C01819=1060.196,-45.835,434.393,171.436,27.271,155.094
C01820=1060.190,-46.085,434.406,171.434,27.269,155.094
C01821=1060.184,-46.335,434.419,171.432,27.267,155.094
C01822=1060.178,-46.584,434.432,171.431,27.265,155.094
C01823=1060.172,-46.833,434.444,171.429,27.263,155.093
C01824=1060.166,-47.083,434.456,171.428,27.261,155.093
C01825=1060.160,-47.332,434.469,171.426,27.259,155.093
C01826=1060.154,-47.582,434.481,171.424,27.257,155.093
C01827=1060.147,-47.831,434.494,171.423,27.255,155.093
C01828=1060.142,-48.081,434.506,171.421,27.254,155.093
C01829=1060.136,-48.331,434.519,171.419,27.251,155.092
C01830=1060.130,-48.581,434.531,171.418,27.250,155.092
C01831=1060.123,-48.831,434.543,171.416,27.247,155.092
C01832=1060.117,-49.080,434.556,171.414,27.246,155.092
C01833=1060.112,-49.330,434.568,171.413,27.244,155.092
C01834=1060.105,-49.579,434.581,171.411,27.242,155.091
C01835=1060.099,-49.828,434.593,171.409,27.240,155.091
C01836=1060.093,-50.108,434.607,171.408,27.238,155.091
C01837=1060.086,-50.387,434.621,171.406,27.236,155.091
C01838=1060.078,-50.667,434.635,171.403,27.234,155.091
C01839=1060.071,-50.946,434.648,171.402,27.232,155.091
C01840=1060.065,-51.195,434.660,171.400,27.230,155.090
C01841=1060.059,-51.444,434.673,171.399,27.228,155.090
C01842=1060.053,-51.694,434.685,171.397,27.227,155.090
C01843=1060.047,-51.944,434.697,171.395,27.225,155.090
C01844=1060.040,-52.193,434.709,171.394,27.223,155.090
C01845=1060.034,-52.443,434.722,171.392,27.221,155.090
C01846=1060.028,-52.693,434.734,171.390,27.219,155.089
C01847=1060.021,-52.942,434.746,171.389,27.218,155.089
C01848=1060.015,-53.192,434.758,171.387,27.216,155.089
C01849=1060.008,-53.442,434.770,171.385,27.214,155.089
C01850=1060.003,-53.691,434.782,171.384,27.213,155.089
C01851=1059.996,-53.941,434.794,171.382,27.211,155.089
C01852=1059.990,-54.190,434.806,171.380,27.209,155.089
C01853=1059.984,-54.440,434.819,171.378,27.207,155.088
C01854=1059.977,-54.690,434.831,171.377,27.206,155.088
C01855=1059.971,-54.940,434.843,171.375,27.203,155.088
C01856=1059.965,-55.189,434.855,171.374,27.202,155.088
C01857=1059.959,-55.438,434.867,171.371,27.200,155.088
C01858=1059.953,-55.688,434.879,171.369,27.198,155.088
C01859=1059.946,-55.938,434.891,171.368,27.196,155.087
C01860=1059.940,-56.188,434.903,171.366,27.195,155.087
C01861=1059.934,-56.437,434.915,171.364,27.193,155.087
C01862=1059.928,-56.686,434.927,171.362,27.191,155.087
C01863=1059.922,-56.936,434.939,171.361,27.190,155.087
C01864=1059.915,-57.186,434.951,171.359,27.188,155.087
C01865=1059.909,-57.435,434.963,171.357,27.186,155.087
C01866=1059.903,-57.686,434.975,171.356,27.184,155.086
C01867=1059.897,-57.935,434.987,171.354,27.183,155.086
C01868=1059.890,-58.184,434.999,171.352,27.181,155.086
C01869=1059.884,-58.434,435.011,171.351,27.179,155.086
C01870=1059.878,-58.684,435.023,171.349,27.178,155.086
C01871=1059.872,-58.933,435.034,171.347,27.176,155.086
C01872=1059.866,-59.183,435.047,171.346,27.174,155.086
C01873=1059.859,-59.433,435.058,171.344,27.172,155.085
C01874=1059.853,-59.682,435.070,171.342,27.171,155.085
C01875=1059.847,-59.931,435.083,171.341,27.169,155.085
C01876=1059.841,-60.182,435.094,171.339,27.167,155.085
C01877=1059.834,-60.431,435.106,171.337,27.166,155.085
C01878=1059.829,-60.681,435.118,171.336,27.164,155.085
C01879=1059.823,-60.930,435.130,171.334,27.162,155.085
C01880=1059.816,-61.180,435.141,171.332,27.161,155.084
C01881=1059.810,-61.430,435.154,171.331,27.159,155.084
C01882=1059.804,-61.680,435.166,171.329,27.157,155.084
C01883=1059.798,-61.929,435.177,171.326,27.155,155.084
C01884=1059.792,-62.179,435.189,171.325,27.153,155.084
C01885=1059.785,-62.429,435.201,171.323,27.152,155.084
C01886=1059.779,-62.677,435.213,171.321,27.150,155.084
C01887=1059.774,-62.928,435.225,171.320,27.148,155.083
C01888=1059.767,-63.178,435.237,171.318,27.147,155.083
C01889=1059.761,-63.426,435.248,171.316,27.145,155.083
C01890=1059.755,-63.677,435.260,171.315,27.143,155.083
C01891=1059.749,-63.926,435.272,171.313,27.141,155.083
C01892=1059.743,-64.175,435.283,171.311,27.140,155.083
C01893=1059.736,-64.426,435.295,171.309,27.138,155.083
C01894=1059.730,-64.675,435.307,171.308,27.136,155.082
C01895=1059.725,-64.925,435.318,171.306,27.135,155.082
C01896=1059.718,-65.174,435.330,171.304,27.134,155.082
C01897=1059.712,-65.424,435.343,171.303,27.132,155.082
C01898=1059.706,-65.674,435.354,171.301,27.130,155.082
C01899=1059.700,-65.923,435.366,171.299,27.128,155.082
C01900=1059.693,-66.204,435.378,171.297,27.126,155.082
C01901=1059.686,-66.484,435.392,171.295,27.125,155.082
C01902=1059.680,-66.765,435.404,171.293,27.123,155.081
C01903=1059.672,-67.045,435.418,171.292,27.121,155.081
C01904=1059.667,-67.295,435.429,171.290,27.120,155.081
C01905=1059.661,-67.545,435.441,171.287,27.118,155.081
C01906=1059.654,-67.794,435.453,171.286,27.116,155.081
C01907=1059.648,-68.044,435.464,171.284,27.114,155.081
C01908=1059.642,-68.293,435.477,171.282,27.112,155.081
C01909=1059.637,-68.543,435.488,171.281,27.111,155.080
C01910=1059.630,-68.793,435.499,171.279,27.109,155.080
C01911=1059.624,-69.042,435.510,171.277,27.107,155.080
C01912=1059.618,-69.292,435.523,171.276,27.106,155.080
C01913=1059.612,-69.542,435.534,171.274,27.104,155.080
C01914=1059.606,-69.791,435.546,171.272,27.103,155.080
C01915=1059.600,-70.041,435.557,171.270,27.101,155.080
C01916=1059.594,-70.291,435.568,171.269,27.099,155.080
C01917=1059.588,-70.541,435.580,171.267,27.098,155.079
C01918=1059.582,-70.790,435.591,171.265,27.097,155.079
C01919=1059.576,-71.040,435.603,171.264,27.095,155.079
C01920=1059.570,-71.289,435.614,171.262,27.093,155.079
C01921=1059.564,-71.539,435.627,171.260,27.091,155.079
C01922=1059.558,-71.788,435.638,171.259,27.090,155.079
C01923=1059.552,-72.039,435.649,171.257,27.089,155.079
C01924=1059.546,-72.288,435.660,171.255,27.087,155.079
C01925=1059.539,-72.538,435.672,171.253,27.085,155.079
C01926=1059.534,-72.787,435.684,171.251,27.083,155.078
C01927=1059.528,-73.037,435.695,171.249,27.082,155.078
C01928=1059.522,-73.287,435.706,171.247,27.080,155.078
C01929=1059.515,-73.536,435.718,171.246,27.079,155.078
C01930=1059.510,-73.786,435.729,171.244,27.077,155.078
C01931=1059.504,-74.036,435.741,171.242,27.076,155.078
C01932=1059.497,-74.285,435.752,171.241,27.074,155.078
C01933=1059.491,-74.535,435.763,171.239,27.072,155.078
C01934=1059.485,-74.784,435.774,171.237,27.071,155.078
C01935=1059.479,-75.034,435.786,171.235,27.070,155.078
C01936=1059.473,-75.283,435.797,171.234,27.068,155.077
C01937=1059.467,-75.534,435.808,171.232,27.067,155.077
C01938=1059.461,-75.783,435.819,171.230,27.065,155.077
C01939=1059.454,-76.033,435.831,171.229,27.064,155.077
C01940=1059.448,-76.282,435.842,171.227,27.062,155.077
C01941=1059.442,-76.532,435.853,171.225,27.061,155.077
C01942=1059.436,-76.782,435.864,171.223,27.059,155.077
C01943=1059.430,-77.031,435.876,171.221,27.057,155.077
C01944=1059.424,-77.281,435.887,171.219,27.056,155.077
C01945=1059.418,-77.531,435.898,171.217,27.054,155.077
C01946=1059.412,-77.781,435.909,171.216,27.053,155.077
C01947=1059.406,-78.031,435.920,171.214,27.052,155.076
C01948=1059.399,-78.280,435.931,171.212,27.051,155.076
C01949=1059.393,-78.530,435.943,171.210,27.049,155.076
C01950=1059.387,-78.779,435.954,171.209,27.048,155.076
C01951=1059.381,-79.030,435.965,171.207,27.046,155.076
C01952=1059.375,-79.279,435.976,171.205,27.045,155.076
C01953=1059.369,-79.528,435.987,171.204,27.043,155.076
C01954=1059.363,-79.778,435.999,171.202,27.042,155.076
C01955=1059.356,-80.027,436.009,171.200,27.040,155.076
C01956=1059.350,-80.277,436.020,171.198,27.039,155.076
C01957=1059.344,-80.527,436.031,171.196,27.037,155.076
C01958=1059.338,-80.777,436.042,171.194,27.036,155.076
C01959=1059.332,-81.026,436.052,171.192,27.035,155.076
C01960=1059.325,-81.277,436.064,171.191,27.033,155.075
C01961=1059.319,-81.526,436.075,171.189,27.032,155.075
C01962=1059.312,-81.776,436.085,171.187,27.031,155.075
C01963=1059.306,-82.025,436.097,171.185,27.029,155.075
C01964=1059.300,-82.308,436.109,171.183,27.028,155.075
C01965=1059.292,-82.590,436.122,171.181,27.026,155.075
C01966=1059.285,-82.873,436.133,171.179,27.025,155.075
C01967=1059.279,-83.156,436.146,171.177,27.023,155.075
C01968=1059.272,-83.405,436.156,171.176,27.022,155.075
C01969=1059.266,-83.655,436.168,171.173,27.021,155.075
C01970=1059.260,-83.905,436.179,171.171,27.019,155.075
C01971=1059.254,-84.154,436.189,171.169,27.018,155.075
C01972=1059.247,-84.404,436.200,171.168,27.017,155.075
C01973=1059.241,-84.654,436.211,171.166,27.015,155.075
C01974=1059.235,-84.904,436.222,171.164,27.014,155.075
C01975=1059.229,-85.153,436.233,171.162,27.013,155.075
C01976=1059.223,-85.403,436.243,171.161,27.012,155.075
C01977=1059.216,-85.653,436.255,171.159,27.010,155.074
C01978=1059.210,-85.902,436.265,171.157,27.009,155.074
C01979=1059.204,-86.152,436.276,171.155,27.008,155.074
C01980=1059.198,-86.402,436.287,171.154,27.007,155.074
C01981=1059.191,-86.651,436.297,171.152,27.005,155.074
C01982=1059.185,-86.901,436.309,171.149,27.004,155.074
C01983=1059.179,-87.151,436.319,171.148,27.002,155.074
C01984=1059.173,-87.400,436.330,171.146,27.001,155.074
C01985=1059.167,-87.651,436.340,171.144,27.000,155.074
C01986=1059.161,-87.900,436.351,171.142,26.998,155.074
C01987=1059.155,-88.149,436.361,171.141,26.997,155.074
C01988=1059.148,-88.399,436.373,171.139,26.996,155.074
C01989=1059.143,-88.649,436.384,171.137,26.994,155.074
C01990=1059.136,-88.898,436.394,171.135,26.993,155.074
C01991=1059.130,-89.148,436.405,171.134,26.992,155.074
C01992=1059.124,-89.398,436.415,171.132,26.991,155.074
C01993=1059.118,-89.648,436.426,171.130,26.990,155.074
C01994=1059.112,-89.897,436.436,171.128,26.989,155.074
C01995=1059.106,-90.147,436.448,171.126,26.987,155.074
C01996=1059.099,-90.396,436.458,171.124,26.986,155.074
C01997=1059.094,-90.646,436.469,171.122,26.985,155.074
C01998=1059.087,-90.896,436.479,171.120,26.983,155.074
C01999=1059.081,-91.146,436.490,171.118,26.982,155.074
C02000=1059.075,-91.395,436.500,171.117,26.981,155.074
C02001=1059.069,-91.645,436.511,171.115,26.980,155.073
C02002=1059.063,-91.895,436.521,171.113,26.978,155.073
C02003=1059.057,-92.145,436.532,171.111,26.977,155.073
C02004=1059.051,-92.394,436.542,171.110,26.976,155.073
C02005=1059.045,-92.644,436.553,171.108,26.975,155.073
C02006=1059.038,-92.894,436.563,171.106,26.974,155.073
C02007=1059.032,-93.144,436.574,171.104,26.973,155.073
C02008=1059.027,-93.393,436.585,171.102,26.971,155.073
C02009=1059.020,-93.642,436.595,171.100,26.970,155.073
C02010=1059.014,-93.893,436.606,171.098,26.969,155.073
C02011=1059.008,-94.142,436.616,171.096,26.967,155.073
C02012=1059.002,-94.392,436.627,171.095,26.966,155.073
C02013=1058.996,-94.642,436.637,171.093,26.965,155.073
C02014=1058.990,-94.891,436.647,171.091,26.964,155.073
C02015=1058.984,-95.141,436.659,171.089,26.963,155.073
C02016=1058.977,-95.391,436.668,171.088,26.962,155.073
C02017=1058.972,-95.640,436.679,171.086,26.961,155.073
C02018=1058.966,-95.890,436.690,171.084,26.959,155.073
C02019=1058.960,-96.140,436.700,171.082,26.958,155.073
C02020=1058.954,-96.389,436.710,171.079,26.957,155.073
C02021=1058.947,-96.639,436.721,171.078,26.956,155.073
C02022=1058.942,-96.889,436.731,171.076,26.955,155.073
C02023=1058.935,-97.138,436.742,171.074,26.954,155.073
C02024=1058.930,-97.388,436.752,171.072,26.952,155.073
C02025=1058.923,-97.638,436.762,171.071,26.951,155.073
C02026=1058.917,-97.887,436.773,171.069,26.950,155.073
C02027=1058.911,-98.138,436.783,171.067,26.949,155.073
C02028=1058.904,-98.422,436.795,171.065,26.948,155.073
C02029=1058.897,-98.707,436.807,171.063,26.947,155.073
C02030=1058.889,-98.993,436.818,171.061,26.945,155.073
C02031=1058.883,-99.277,436.830,171.058,26.944,155.073
C02032=1058.876,-99.526,436.840,171.056,26.943,155.073
C02033=1058.871,-99.777,436.850,171.055,26.942,155.073
C02034=1058.864,-100.026,436.860,171.053,26.941,155.073
C02035=1058.858,-100.276,436.870,171.051,26.939,155.073
C02036=1058.852,-100.526,436.881,171.049,26.939,155.073
C02037=1058.846,-100.776,436.891,171.047,26.938,155.073
C02038=1058.839,-101.025,436.901,171.046,26.937,155.073
C02039=1058.834,-101.275,436.911,171.044,26.936,155.073
C02040=1058.827,-101.524,436.921,171.042,26.934,155.073
C02041=1058.821,-101.774,436.931,171.040,26.934,155.073
C02042=1058.815,-102.025,436.942,171.037,26.933,155.073
C02043=1058.809,-102.274,436.952,171.036,26.931,155.073
C02044=1058.802,-102.524,436.961,171.034,26.930,155.073
C02045=1058.797,-102.773,436.972,171.032,26.929,155.073
C02046=1058.790,-103.023,436.982,171.030,26.929,155.073
C02047=1058.784,-103.272,436.992,171.028,26.927,155.073
C02048=1058.779,-103.522,437.002,171.027,26.926,155.073
C02049=1058.772,-103.772,437.012,171.025,26.925,155.073
C02050=1058.766,-104.021,437.022,171.023,26.925,155.073
C02051=1058.760,-104.272,437.033,171.021,26.924,155.073
C02052=1058.754,-104.522,437.042,171.019,26.922,155.073
C02053=1058.747,-104.771,437.052,171.018,26.922,155.073
C02054=1058.741,-105.021,437.062,171.015,26.920,155.073
C02055=1058.735,-105.270,437.073,171.013,26.919,155.073
C02056=1058.729,-105.520,437.082,171.011,26.918,155.073
C02057=1058.723,-105.770,437.092,171.009,26.918,155.073
C02058=1058.716,-106.019,437.102,171.008,26.917,155.073
C02059=1058.711,-106.269,437.113,171.006,26.915,155.073
C02060=1058.705,-106.519,437.122,171.004,26.915,155.073
C02061=1058.699,-106.769,437.132,171.002,26.914,155.073
C02062=1058.692,-107.018,437.142,171.000,26.913,155.073
C02063=1058.687,-107.268,437.152,170.999,26.912,155.073
C02064=1058.681,-107.518,437.162,170.997,26.911,155.073
C02065=1058.674,-107.767,437.172,170.994,26.910,155.073
C02066=1058.668,-108.017,437.182,170.992,26.909,155.073
C02067=1058.661,-108.267,437.191,170.990,26.908,155.073
C02068=1058.655,-108.517,437.201,170.989,26.907,155.073
C02069=1058.649,-108.766,437.211,170.987,26.906,155.073
C02070=1058.643,-109.016,437.221,170.985,26.906,155.073
C02071=1058.637,-109.266,437.231,170.983,26.905,155.073
C02072=1058.631,-109.516,437.241,170.981,26.904,155.073
C02073=1058.625,-109.766,437.250,170.979,26.903,155.073
C02074=1058.618,-110.015,437.260,170.978,26.902,155.074
C02075=1058.612,-110.265,437.270,170.976,26.901,155.073
C02076=1058.606,-110.514,437.280,170.973,26.900,155.074
C02077=1058.600,-110.764,437.289,170.971,26.899,155.074
C02078=1058.594,-111.014,437.299,170.969,26.899,155.074
C02079=1058.588,-111.264,437.309,170.968,26.898,155.074
C02080=1058.582,-111.513,437.319,170.966,26.897,155.074
C02081=1058.575,-111.763,437.329,170.964,26.896,155.074
C02082=1058.569,-112.013,437.338,170.962,26.895,155.074
C02083=1058.563,-112.263,437.348,170.960,26.894,155.074
C02084=1058.557,-112.513,437.357,170.958,26.894,155.074
C02085=1058.551,-112.762,437.367,170.957,26.893,155.074
C02086=1058.544,-113.012,437.377,170.955,26.892,155.074
C02087=1058.538,-113.262,437.386,170.953,26.891,155.074
C02088=1058.532,-113.511,437.396,170.950,26.890,155.074
C02089=1058.526,-113.761,437.407,170.948,26.890,155.074
C02090=1058.520,-114.011,437.416,170.946,26.889,155.074
C02091=1058.515,-114.260,437.425,170.945,26.888,155.074
C02092=1058.507,-114.543,437.436,170.943,26.887,155.074
C02093=1058.500,-114.827,437.447,170.940,26.886,155.074
C02094=1058.493,-115.111,437.458,170.938,26.886,155.075
C02095=1058.486,-115.394,437.469,170.936,26.884,155.074
C02096=1058.480,-115.644,437.478,170.934,26.884,155.075
C02097=1058.474,-115.894,437.488,170.933,26.883,155.075
C02098=1058.468,-116.144,437.497,170.930,26.882,155.075
C02099=1058.462,-116.393,437.507,170.928,26.881,155.075
C02100=1058.456,-116.643,437.516,170.926,26.881,155.075
C02101=1058.450,-116.892,437.526,170.924,26.880,155.075
C02102=1058.443,-117.142,437.535,170.922,26.879,155.075
C02103=1058.437,-117.392,437.544,170.920,26.879,155.075
C02104=1058.431,-117.641,437.554,170.919,26.878,155.075
C02105=1058.425,-117.891,437.563,170.917,26.877,155.075
C02106=1058.418,-118.141,437.573,170.915,26.876,155.075
C02107=1058.412,-118.391,437.582,170.913,26.876,155.075
C02108=1058.406,-118.641,437.592,170.911,26.875,155.075
C02109=1058.400,-118.890,437.602,170.908,26.874,155.075
C02110=1058.394,-119.140,437.611,170.907,26.873,155.076
C02111=1058.388,-119.390,437.621,170.905,26.873,155.076
C02112=1058.382,-119.639,437.630,170.903,26.872,155.076
C02113=1058.376,-119.889,437.639,170.901,26.871,155.076
C02114=1058.369,-120.139,437.648,170.899,26.871,155.076
C02115=1058.363,-120.389,437.657,170.897,26.870,155.076
C02116=1058.357,-120.639,437.667,170.895,26.870,155.076
C02117=1058.351,-120.888,437.676,170.894,26.868,155.076
C02118=1058.345,-121.138,437.686,170.892,26.868,155.076
C02119=1058.339,-121.387,437.695,170.890,26.867,155.076
C02120=1058.333,-121.637,437.705,170.888,26.867,155.076
C02121=1058.327,-121.888,437.714,170.885,26.866,155.076
C02122=1058.320,-122.137,437.723,170.883,26.866,155.077
C02123=1058.314,-122.387,437.732,170.881,26.865,155.077
C02124=1058.308,-122.637,437.742,170.880,26.864,155.077
C02125=1058.302,-122.886,437.751,170.878,26.863,155.077
C02126=1058.296,-123.136,437.760,170.876,26.863,155.077
C02127=1058.290,-123.386,437.769,170.874,26.862,155.077
C02128=1058.283,-123.635,437.778,170.872,26.862,155.077
C02129=1058.277,-123.885,437.788,170.870,26.861,155.077
C02130=1058.271,-124.135,437.797,170.868,26.861,155.077
C02131=1058.266,-124.385,437.806,170.866,26.860,155.077
C02132=1058.259,-124.635,437.816,170.864,26.859,155.077
C02133=1058.252,-124.884,437.824,170.862,26.859,155.078
C02134=1058.246,-125.134,437.834,170.860,26.858,155.078
C02135=1058.240,-125.384,437.843,170.858,26.858,155.078
C02136=1058.235,-125.633,437.852,170.856,26.857,155.078
C02137=1058.228,-125.883,437.861,170.854,26.857,155.078
C02138=1058.222,-126.133,437.870,170.852,26.856,155.078
C02139=1058.216,-126.383,437.880,170.850,26.856,155.078
C02140=1058.210,-126.633,437.889,170.849,26.855,155.078
C02141=1058.204,-126.882,437.897,170.847,26.855,155.078
C02142=1058.198,-127.132,437.907,170.845,26.854,155.078
C02143=1058.191,-127.382,437.916,170.843,26.853,155.078
C02144=1058.185,-127.632,437.924,170.840,26.853,155.079
C02145=1058.179,-127.882,437.934,170.838,26.852,155.079
C02146=1058.174,-128.131,437.944,170.836,26.851,155.079
C02147=1058.171,-128.382,437.954,170.835,26.849,155.079
C02148=1058.168,-128.632,437.966,170.833,26.847,155.078
C02149=1058.168,-128.883,437.977,170.833,26.844,155.078
C02150=1058.169,-129.133,437.990,170.831,26.841,155.078
C02151=1058.170,-129.383,438.003,170.830,26.837,155.077
C02152=1058.173,-129.635,438.017,170.830,26.833,155.076
C02153=1058.177,-129.886,438.032,170.829,26.827,155.075
C02154=1058.183,-130.137,438.048,170.828,26.822,155.075
C02155=1058.190,-130.387,438.063,170.828,26.816,155.073
C02156=1057.814,-130.410,437.863,170.780,26.978,155.107
C02157=1057.807,-130.160,437.846,170.781,26.984,155.108
C02158=1057.802,-129.909,437.831,170.781,26.990,155.109
C02159=1057.797,-129.658,437.817,170.782,26.995,155.109
C02160=1057.794,-129.406,437.803,170.782,26.999,155.110
C02161=1057.791,-129.156,437.789,170.783,27.003,155.111
C02162=1057.791,-128.906,437.776,170.785,27.006,155.111
C02163=1057.792,-128.656,437.764,170.786,27.009,155.112
C02164=1057.795,-128.405,437.754,170.788,27.012,155.112
C02165=1057.798,-128.155,437.743,170.789,27.013,155.112
C02166=1057.803,-127.905,437.733,170.791,27.015,155.112
C02167=1057.809,-127.655,437.724,170.793,27.015,155.112
C02168=1057.815,-127.405,437.714,170.795,27.016,155.112
C02169=1057.821,-127.154,437.705,170.797,27.016,155.112
C02170=1057.826,-126.905,437.696,170.799,27.017,155.112
C02171=1057.833,-126.656,437.687,170.801,27.017,155.111
C02172=1057.839,-126.405,437.678,170.803,27.018,155.111
C02173=1057.845,-126.156,437.669,170.804,27.018,155.111
C02174=1057.852,-125.906,437.660,170.806,27.019,155.111
C02175=1057.858,-125.656,437.651,170.808,27.019,155.111
C02176=1057.864,-125.407,437.642,170.810,27.020,155.111
C02177=1057.870,-125.157,437.632,170.813,27.021,155.111
C02178=1057.877,-124.907,437.623,170.815,27.021,155.111
C02179=1057.883,-124.657,437.614,170.817,27.022,155.111
C02180=1057.888,-124.408,437.605,170.819,27.022,155.111
C02181=1057.894,-124.158,437.596,170.820,27.023,155.110
C02182=1057.901,-123.909,437.587,170.822,27.023,155.110
C02183=1057.907,-123.658,437.578,170.824,27.024,155.110
C02184=1057.913,-123.408,437.568,170.826,27.024,155.110
C02185=1057.919,-123.159,437.559,170.828,27.025,155.110
C02186=1057.925,-122.910,437.550,170.830,27.025,155.110
C02187=1057.931,-122.660,437.540,170.832,27.026,155.110
C02188=1057.938,-122.410,437.532,170.835,27.027,155.110
C02189=1057.944,-122.160,437.522,170.836,27.028,155.110
C02190=1057.950,-121.910,437.513,170.838,27.028,155.110
C02191=1057.956,-121.661,437.503,170.840,27.029,155.110
C02192=1057.962,-121.411,437.494,170.842,27.029,155.109
C02193=1057.968,-121.161,437.485,170.844,27.030,155.109
C02194=1057.974,-120.911,437.475,170.846,27.030,155.109
C02195=1057.980,-120.661,437.466,170.848,27.031,155.109
C02196=1057.987,-120.412,437.457,170.849,27.032,155.109
C02197=1057.993,-120.162,437.447,170.851,27.033,155.109
C02198=1057.999,-119.912,437.438,170.853,27.033,155.109
C02199=1058.005,-119.663,437.429,170.856,27.034,155.109
C02200=1058.011,-119.413,437.419,170.858,27.034,155.109
C02201=1058.017,-119.163,437.409,170.860,27.035,155.109
C02202=1058.023,-118.913,437.401,170.862,27.036,155.109
C02203=1058.029,-118.663,437.391,170.863,27.037,155.109
C02204=1058.036,-118.413,437.381,170.865,27.037,155.109
C02205=1058.042,-118.164,437.372,170.867,27.038,155.109
C02206=1058.049,-117.914,437.363,170.869,27.039,155.108
C02207=1058.055,-117.664,437.353,170.871,27.039,155.108
C02208=1058.060,-117.415,437.344,170.873,27.040,155.108
C02209=1058.067,-117.165,437.335,170.875,27.041,155.108
C02210=1058.073,-116.916,437.325,170.877,27.042,155.108
C02211=1058.079,-116.666,437.315,170.879,27.042,155.108
C02212=1058.085,-116.416,437.306,170.881,27.043,155.108
C02213=1058.091,-116.166,437.296,170.883,27.044,155.108
C02214=1058.097,-115.916,437.287,170.885,27.044,155.108
C02215=1058.104,-115.667,437.277,170.887,27.045,155.108
C02216=1058.110,-115.417,437.268,170.888,27.046,155.108
C02217=1058.117,-115.133,437.257,170.891,27.047,155.108
C02218=1058.123,-114.850,437.246,170.893,27.047,155.108
C02219=1058.131,-114.566,437.235,170.895,27.048,155.108
C02220=1058.138,-114.283,437.224,170.898,27.049,155.107
C02221=1058.143,-114.034,437.215,170.900,27.050,155.107
C02222=1058.150,-113.784,437.205,170.901,27.051,155.107
C02223=1058.156,-113.535,437.195,170.903,27.051,155.107
C02224=1058.162,-113.285,437.186,170.905,27.053,155.107
C02225=1058.168,-113.035,437.176,170.907,27.053,155.107
C02226=1058.174,-112.785,437.166,170.909,27.054,155.107
C02227=1058.180,-112.535,437.156,170.911,27.055,155.107
C02228=1058.186,-112.285,437.147,170.912,27.056,155.107
C02229=1058.192,-112.035,437.137,170.915,27.057,155.107
C02230=1058.199,-111.786,437.128,170.917,27.058,155.107
C02231=1058.205,-111.536,437.117,170.919,27.058,155.107
C02232=1058.211,-111.287,437.108,170.921,27.059,155.107
C02233=1058.217,-111.037,437.098,170.923,27.060,155.107
C02234=1058.224,-110.787,437.089,170.924,27.061,155.107
C02235=1058.230,-110.537,437.079,170.926,27.062,155.107
C02236=1058.235,-110.287,437.069,170.928,27.062,155.107
C02237=1058.242,-110.038,437.059,170.930,27.063,155.107
C02238=1058.248,-109.788,437.049,170.932,27.064,155.107
C02239=1058.254,-109.538,437.040,170.934,27.065,155.107
C02240=1058.260,-109.289,437.030,170.936,27.066,155.107
C02241=1058.266,-109.039,437.020,170.938,27.067,155.107
C02242=1058.273,-108.790,437.010,170.940,27.068,155.107
C02243=1058.279,-108.540,437.001,170.942,27.068,155.106
C02244=1058.284,-108.290,436.990,170.944,27.070,155.107
C02245=1058.291,-108.039,436.980,170.946,27.070,155.106
C02246=1058.298,-107.790,436.970,170.947,27.071,155.106
C02247=1058.304,-107.540,436.961,170.949,27.072,155.106
C02248=1058.310,-107.290,436.951,170.951,27.073,155.106
C02249=1058.316,-107.041,436.941,170.953,27.074,155.106
C02250=1058.322,-106.791,436.931,170.955,27.075,155.106
C02251=1058.328,-106.541,436.921,170.957,27.076,155.106
C02252=1058.334,-106.292,436.911,170.959,27.077,155.106
C02253=1058.341,-106.042,436.901,170.961,27.078,155.106
C02254=1058.346,-105.792,436.891,170.963,27.079,155.106
C02255=1058.352,-105.542,436.881,170.965,27.080,155.106
C02256=1058.359,-105.293,436.871,170.966,27.080,155.106
C02257=1058.365,-105.043,436.862,170.968,27.081,155.106
C02258=1058.370,-104.793,436.851,170.970,27.083,155.106
C02259=1058.377,-104.544,436.841,170.972,27.083,155.106
C02260=1058.383,-104.294,436.832,170.974,27.084,155.106
C02261=1058.389,-104.044,436.821,170.975,27.085,155.106
C02262=1058.396,-103.794,436.811,170.978,27.086,155.106
C02263=1058.402,-103.545,436.801,170.980,27.087,155.106
C02264=1058.408,-103.295,436.791,170.982,27.088,155.106
C02265=1058.414,-103.045,436.781,170.984,27.089,155.106
C02266=1058.420,-102.796,436.771,170.986,27.090,155.106
C02267=1058.426,-102.546,436.761,170.987,27.091,155.106
C02268=1058.432,-102.296,436.751,170.989,27.092,155.106
C02269=1058.438,-102.047,436.740,170.991,27.093,155.106
C02270=1058.445,-101.797,436.731,170.993,27.094,155.106
C02271=1058.451,-101.547,436.720,170.995,27.095,155.106
C02272=1058.457,-101.297,436.710,170.996,27.096,155.106
C02273=1058.463,-101.048,436.700,170.999,27.098,155.106
C02274=1058.469,-100.798,436.690,171.001,27.099,155.106
C02275=1058.475,-100.549,436.679,171.003,27.100,155.106
C02276=1058.481,-100.299,436.670,171.005,27.100,155.106
C02277=1058.488,-100.049,436.659,171.006,27.101,155.106
C02278=1058.494,-99.799,436.649,171.008,27.103,155.106
C02279=1058.500,-99.550,436.639,171.010,27.104,155.106
C02280=1058.506,-99.300,436.629,171.012,27.105,155.106
C02281=1058.513,-99.015,436.617,171.014,27.106,155.106
C02282=1058.520,-98.729,436.606,171.016,27.107,155.106
C02283=1058.527,-98.445,436.594,171.018,27.108,155.106
C02284=1058.534,-98.159,436.581,171.021,27.110,155.106
C02285=1058.541,-97.910,436.572,171.023,27.110,155.106
C02286=1058.547,-97.660,436.562,171.024,27.111,155.106
C02287=1058.553,-97.411,436.551,171.026,27.113,155.106
C02288=1058.559,-97.161,436.541,171.028,27.114,155.106
C02289=1058.565,-96.912,436.530,171.030,27.115,155.106
C02290=1058.571,-96.661,436.520,171.031,27.116,155.106
C02291=1058.577,-96.412,436.509,171.033,27.117,155.106
C02292=1058.583,-96.162,436.499,171.035,27.118,155.106
C02293=1058.589,-95.912,436.489,171.037,27.119,155.106
C02294=1058.595,-95.663,436.478,171.040,27.121,155.106
C02295=1058.602,-95.413,436.467,171.041,27.122,155.106
C02296=1058.607,-95.163,436.457,171.043,27.123,155.106
C02297=1058.613,-94.913,436.446,171.045,27.125,155.106
C02298=1058.620,-94.664,436.436,171.047,27.126,155.106
C02299=1058.625,-94.414,436.426,171.048,27.127,155.106
C02300=1058.632,-94.164,436.415,171.050,27.128,155.106
C02301=1058.638,-93.915,436.404,171.052,27.129,155.106
C02302=1058.643,-93.665,436.394,171.054,27.130,155.106
C02303=1058.650,-93.415,436.384,171.055,27.131,155.106
C02304=1058.656,-93.166,436.373,171.057,27.132,155.106
C02305=1058.663,-92.916,436.362,171.059,27.134,155.106
C02306=1058.668,-92.666,436.352,171.062,27.135,155.106
C02307=1058.674,-92.417,436.341,171.064,27.136,155.106
C02308=1058.680,-92.167,436.331,171.065,27.138,155.107
C02309=1058.687,-91.917,436.320,171.067,27.139,155.107
C02310=1058.692,-91.667,436.310,171.069,27.140,155.107
C02311=1058.699,-91.418,436.299,171.071,27.141,155.107
C02312=1058.704,-91.168,436.289,171.072,27.142,155.107
C02313=1058.711,-90.918,436.278,171.074,27.143,155.107
C02314=1058.717,-90.668,436.268,171.076,27.144,155.107
C02315=1058.723,-90.419,436.257,171.078,27.146,155.107
C02316=1058.730,-90.169,436.246,171.079,27.147,155.107
C02317=1058.735,-89.920,436.235,171.081,27.148,155.107
C02318=1058.741,-89.670,436.224,171.084,27.150,155.107
C02319=1058.748,-89.421,436.214,171.086,27.151,155.107
C02320=1058.754,-89.170,436.204,171.087,27.152,155.107
C02321=1058.759,-88.921,436.193,171.089,27.154,155.107
C02322=1058.766,-88.671,436.183,171.091,27.155,155.107
C02323=1058.772,-88.421,436.171,171.093,27.156,155.107
C02324=1058.778,-88.172,436.160,171.094,27.157,155.107
C02325=1058.784,-87.923,436.150,171.096,27.158,155.107
C02326=1058.791,-87.672,436.139,171.098,27.160,155.107
C02327=1058.797,-87.423,436.129,171.100,27.161,155.107
C02328=1058.803,-87.173,436.118,171.101,27.162,155.107
C02329=1058.809,-86.923,436.107,171.103,27.163,155.107
C02330=1058.815,-86.673,436.096,171.105,27.165,155.108
C02331=1058.821,-86.424,436.086,171.108,27.166,155.108
C02332=1058.828,-86.174,436.075,171.109,27.167,155.108
C02333=1058.833,-85.924,436.064,171.111,27.169,155.108
C02334=1058.840,-85.675,436.053,171.113,27.170,155.108
C02335=1058.846,-85.425,436.042,171.115,27.171,155.108
C02336=1058.852,-85.176,436.031,171.116,27.173,155.108
C02337=1058.859,-84.926,436.021,171.118,27.174,155.108
C02338=1058.865,-84.676,436.010,171.120,27.175,155.108
C02339=1058.870,-84.427,435.999,171.122,27.176,155.108
C02340=1058.877,-84.177,435.988,171.124,27.178,155.108
C02341=1058.883,-83.927,435.978,171.125,27.179,155.108
C02342=1058.890,-83.677,435.966,171.127,27.180,155.108
C02343=1058.895,-83.428,435.955,171.130,27.182,155.108
C02344=1058.902,-83.178,435.945,171.131,27.183,155.108
C02345=1058.909,-82.895,435.932,171.133,27.185,155.108
C02346=1058.916,-82.613,435.920,171.135,27.186,155.108
C02347=1058.923,-82.331,435.908,171.138,27.188,155.108
C02348=1058.930,-82.047,435.896,171.139,27.189,155.108
C02349=1058.936,-81.798,435.884,171.141,27.191,155.109
C02350=1058.943,-81.548,435.874,171.143,27.192,155.109
C02351=1058.949,-81.298,435.862,171.145,27.193,155.109
C02352=1058.955,-81.049,435.851,171.146,27.194,155.109
C02353=1058.962,-80.799,435.841,171.148,27.196,155.109
C02354=1058.968,-80.549,435.830,171.150,27.197,155.109
C02355=1058.974,-80.299,435.819,171.152,27.199,155.109
C02356=1058.980,-80.050,435.808,171.154,27.200,155.109
C02357=1058.987,-79.800,435.797,171.156,27.201,155.109
C02358=1058.992,-79.550,435.786,171.158,27.203,155.109
C02359=1058.999,-79.301,435.774,171.160,27.204,155.109
C02360=1059.005,-79.051,435.763,171.161,27.205,155.109
C02361=1059.011,-78.802,435.753,171.163,27.207,155.109
C02362=1059.017,-78.552,435.741,171.165,27.208,155.109
C02363=1059.023,-78.302,435.730,171.166,27.209,155.109
C02364=1059.029,-78.053,435.718,171.168,27.211,155.110
C02365=1059.035,-77.803,435.708,171.170,27.213,155.110
C02366=1059.041,-77.553,435.696,171.172,27.214,155.110
C02367=1059.047,-77.303,435.685,171.173,27.216,155.110
C02368=1059.054,-77.053,435.674,171.175,27.217,155.110
C02369=1059.060,-76.804,435.663,171.178,27.219,155.110
C02370=1059.066,-76.554,435.651,171.179,27.220,155.110
C02371=1059.072,-76.305,435.641,171.181,27.222,155.110
C02372=1059.078,-76.054,435.629,171.183,27.223,155.110
C02373=1059.084,-75.806,435.618,171.185,27.224,155.110
C02374=1059.090,-75.555,435.606,171.186,27.226,155.111
C02375=1059.096,-75.306,435.596,171.188,27.227,155.111
C02376=1059.103,-75.056,435.584,171.190,27.229,155.111
C02377=1059.108,-74.807,435.573,171.192,27.230,155.111
C02378=1059.115,-74.557,435.561,171.193,27.232,155.111
C02379=1059.121,-74.307,435.551,171.195,27.233,155.111
C02380=1059.127,-74.058,435.539,171.197,27.235,155.111
C02381=1059.133,-73.808,435.528,171.198,27.236,155.111
C02382=1059.139,-73.558,435.517,171.200,27.238,155.111
C02383=1059.145,-73.309,435.505,171.202,27.239,155.111
C02384=1059.152,-73.059,435.494,171.204,27.241,155.111
C02385=1059.157,-72.809,435.483,171.206,27.243,155.112
C02386=1059.163,-72.559,435.470,171.208,27.244,155.112
C02387=1059.169,-72.310,435.459,171.210,27.246,155.112
C02388=1059.176,-72.060,435.447,171.211,27.247,155.112
C02389=1059.181,-71.811,435.437,171.213,27.249,155.112
C02390=1059.188,-71.561,435.425,171.215,27.251,155.112
C02391=1059.193,-71.312,435.413,171.216,27.252,155.112
C02392=1059.199,-71.061,435.402,171.218,27.253,155.112
C02393=1059.205,-70.813,435.390,171.220,27.255,155.112
C02394=1059.212,-70.562,435.379,171.222,27.257,155.113
C02395=1059.217,-70.313,435.367,171.223,27.259,155.113
C02396=1059.223,-70.063,435.356,171.225,27.260,155.113
C02397=1059.230,-69.813,435.344,171.227,27.261,155.113
C02398=1059.236,-69.564,435.333,171.228,27.263,155.113
C02399=1059.243,-69.314,435.321,171.230,27.265,155.113
C02400=1059.248,-69.064,435.309,171.232,27.266,155.113
C02401=1059.254,-68.815,435.297,171.233,27.268,155.114
C02402=1059.260,-68.565,435.286,171.235,27.270,155.114
C02403=1059.267,-68.316,435.275,171.237,27.271,155.114
C02404=1059.272,-68.065,435.263,171.239,27.273,155.114
C02405=1059.278,-67.816,435.251,171.241,27.275,155.114
C02406=1059.285,-67.566,435.240,171.243,27.276,155.114
C02407=1059.291,-67.317,435.228,171.245,27.278,155.114
C02408=1059.296,-67.067,435.216,171.246,27.280,155.114
C02409=1059.303,-66.787,435.203,171.248,27.281,155.115
C02410=1059.310,-66.506,435.191,171.250,27.283,155.115
C02411=1059.317,-66.226,435.177,171.252,27.285,155.115
C02412=1059.324,-65.945,435.164,171.254,27.287,155.115
C02413=1059.330,-65.696,435.152,171.256,27.289,155.115
C02414=1059.335,-65.446,435.141,171.257,27.290,155.115
C02415=1059.342,-65.196,435.129,171.259,27.292,155.115
C02416=1059.349,-64.947,435.117,171.261,27.294,155.115
C02417=1059.354,-64.697,435.106,171.262,27.295,155.116
C02418=1059.360,-64.447,435.093,171.264,27.296,155.116
C02419=1059.367,-64.197,435.082,171.266,27.298,155.116
C02420=1059.373,-63.948,435.070,171.268,27.300,155.116
C02421=1059.378,-63.698,435.058,171.269,27.302,155.116
C02422=1059.385,-63.448,435.047,171.271,27.303,155.116
C02423=1059.391,-63.199,435.035,171.273,27.305,155.116
C02424=1059.398,-62.950,435.023,171.274,27.307,155.116
C02425=1059.403,-62.699,435.011,171.276,27.308,155.117
C02426=1059.409,-62.450,435.000,171.279,27.310,155.117
C02427=1059.416,-62.201,434.988,171.280,27.312,155.117
C02428=1059.422,-61.951,434.975,171.282,27.314,155.117
C02429=1059.427,-61.701,434.964,171.284,27.315,155.117
C02430=1059.434,-61.452,434.952,171.285,27.317,155.117
C02431=1059.440,-61.202,434.940,171.287,27.319,155.117
C02432=1059.446,-60.952,434.929,171.289,27.321,155.118
C02433=1059.452,-60.703,434.917,171.290,27.322,155.118
C02434=1059.458,-60.453,434.904,171.292,27.324,155.118
C02435=1059.465,-60.203,434.892,171.294,27.326,155.118
C02436=1059.472,-59.954,434.881,171.296,27.327,155.118
C02437=1059.477,-59.704,434.869,171.297,27.329,155.118
C02438=1059.483,-59.454,434.857,171.299,27.331,155.118
C02439=1059.490,-59.205,434.845,171.301,27.332,155.119
C02440=1059.496,-58.955,434.833,171.302,27.334,155.119
C02441=1059.502,-58.706,434.822,171.304,27.336,155.119
C02442=1059.508,-58.456,434.810,171.306,27.338,155.119
C02443=1059.514,-58.206,434.797,171.307,27.339,155.119
C02444=1059.521,-57.957,434.785,171.309,27.341,155.119
C02445=1059.527,-57.708,434.774,171.311,27.343,155.119
C02446=1059.533,-57.458,434.761,171.312,27.344,155.120
C02447=1059.539,-57.208,434.749,171.314,27.346,155.120
C02448=1059.545,-56.958,434.737,171.316,27.348,155.120
C02449=1059.552,-56.708,434.725,171.317,27.349,155.120
C02450=1059.558,-56.459,434.714,171.319,27.351,155.120
C02451=1059.564,-56.209,434.701,171.322,27.353,155.120
C02452=1059.570,-55.960,434.689,171.323,27.355,155.120
C02453=1059.577,-55.710,434.677,171.325,27.356,155.121
C02454=1059.583,-55.460,434.665,171.327,27.358,155.121
C02455=1059.589,-55.211,434.653,171.329,27.360,155.121
C02456=1059.595,-54.962,434.641,171.330,27.362,155.121
C02457=1059.601,-54.711,434.629,171.332,27.363,155.121
C02458=1059.608,-54.462,434.617,171.334,27.365,155.121
C02459=1059.614,-54.212,434.605,171.335,27.367,155.121
C02460=1059.620,-53.962,434.593,171.337,27.368,155.122
C02461=1059.626,-53.712,434.580,171.339,27.370,155.122
C02462=1059.633,-53.463,434.568,171.340,27.372,155.122
C02463=1059.639,-53.214,434.557,171.342,27.374,155.122
C02464=1059.645,-52.964,434.544,171.344,27.376,155.122
C02465=1059.651,-52.715,434.532,171.345,27.377,155.122
C02466=1059.657,-52.465,434.520,171.347,27.379,155.123
C02467=1059.664,-52.215,434.508,171.349,27.381,155.123
C02468=1059.671,-51.966,434.496,171.350,27.383,155.123
C02469=1059.677,-51.716,434.483,171.352,27.384,155.123
C02470=1059.683,-51.466,434.471,171.354,27.386,155.123
C02471=1059.689,-51.216,434.459,171.356,27.388,155.123
C02472=1059.696,-50.967,434.447,171.357,27.390,155.124
C02473=1059.703,-50.688,434.433,171.359,27.392,155.124
C02474=1059.710,-50.409,434.419,171.361,27.394,155.124
C02475=1059.716,-50.130,434.405,171.363,27.396,155.124
C02476=1059.723,-49.851,434.391,171.365,27.398,155.124
C02477=1059.729,-49.601,434.379,171.366,27.400,155.125
C02478=1059.735,-49.351,434.366,171.368,27.401,155.125
C02479=1059.742,-49.101,434.354,171.370,27.403,155.125
C02480=1059.748,-48.852,434.342,171.371,27.405,155.125
C02481=1059.753,-48.602,434.329,171.373,27.407,155.125
C02482=1059.760,-48.353,434.317,171.375,27.409,155.125
C02483=1059.765,-48.103,434.305,171.376,27.411,155.126
C02484=1059.772,-47.854,434.292,171.378,27.413,155.126
C02485=1059.778,-47.604,434.279,171.380,27.415,155.126
C02486=1059.784,-47.354,434.267,171.381,27.417,155.126
C02487=1059.790,-47.104,434.255,171.383,27.419,155.126
C02488=1059.796,-46.854,434.242,171.385,27.421,155.127
C02489=1059.802,-46.605,434.229,171.386,27.422,155.127
C02490=1059.809,-46.356,434.217,171.388,27.424,155.127
C02491=1059.815,-46.106,434.204,171.390,27.426,155.127
C02492=1059.820,-45.857,434.192,171.391,27.428,155.127
C02493=1059.826,-45.607,434.179,171.393,27.430,155.128
C02494=1059.833,-45.358,434.167,171.394,27.432,155.128
C02495=1059.839,-45.108,434.154,171.396,27.434,155.128
C02496=1059.845,-44.858,434.142,171.398,27.436,155.128
C02497=1059.851,-44.608,434.129,171.399,27.438,155.128
C02498=1059.858,-44.359,434.116,171.401,27.439,155.128
C02499=1059.864,-44.109,434.104,171.403,27.442,155.129
C02500=1059.869,-43.859,434.091,171.404,27.443,155.129
C02501=1059.876,-43.610,434.078,171.406,27.446,155.129
C02502=1059.882,-43.361,434.066,171.409,27.448,155.129
C02503=1059.888,-43.111,434.054,171.410,27.449,155.129
C02504=1059.894,-42.861,434.040,171.412,27.452,155.130
C02505=1059.900,-42.612,434.028,171.414,27.453,155.130
C02506=1059.906,-42.362,434.015,171.415,27.456,155.130
C02507=1059.913,-42.113,434.003,171.417,27.457,155.130
C02508=1059.919,-41.863,433.990,171.419,27.460,155.130
C02509=1059.925,-41.613,433.977,171.420,27.461,155.131
C02510=1059.931,-41.364,433.964,171.422,27.463,155.131
C02511=1059.937,-41.114,433.952,171.424,27.465,155.131
C02512=1059.944,-40.864,433.940,171.425,27.467,155.131
C02513=1059.950,-40.615,433.926,171.427,27.469,155.131
C02514=1059.956,-40.365,433.914,171.429,27.471,155.132
C02515=1059.962,-40.116,433.901,171.430,27.473,155.132
C02516=1059.968,-39.866,433.888,171.432,27.475,155.132
C02517=1059.975,-39.616,433.876,171.433,27.477,155.132
C02518=1059.981,-39.367,433.863,171.435,27.479,155.132
C02519=1059.987,-39.117,433.850,171.437,27.481,155.132
C02520=1059.993,-38.868,433.837,171.438,27.483,155.133
C02521=1059.999,-38.618,433.824,171.440,27.484,155.133
C02522=1060.005,-38.369,433.811,171.442,27.487,155.133
C02523=1060.011,-38.119,433.799,171.442,27.489,155.133
C02524=1060.017,-37.870,433.785,171.444,27.490,155.134
C02525=1060.023,-37.620,433.773,171.446,27.493,155.134
C02526=1060.029,-37.370,433.759,171.447,27.494,155.134
C02527=1060.035,-37.121,433.747,171.449,27.497,155.134
C02528=1060.042,-36.871,433.734,171.451,27.499,155.135
C02529=1060.047,-36.621,433.721,171.452,27.501,155.135
C02530=1060.054,-36.371,433.707,171.454,27.503,155.135
C02531=1060.060,-36.122,433.695,171.456,27.505,155.135
C02532=1060.066,-35.872,433.682,171.457,27.507,155.135
C02533=1060.072,-35.622,433.669,171.459,27.509,155.136
C02534=1060.078,-35.373,433.656,171.460,27.511,155.136
C02535=1060.084,-35.123,433.643,171.462,27.513,155.136
C02536=1060.091,-34.874,433.630,171.464,27.515,155.136
C02537=1060.097,-34.595,433.615,171.466,27.518,155.137
C02538=1060.105,-34.316,433.601,171.468,27.520,155.137
C02539=1060.111,-34.038,433.586,171.470,27.522,155.137
C02540=1060.117,-33.759,433.572,171.471,27.524,155.137
C02541=1060.123,-33.510,433.559,171.473,27.526,155.137
C02542=1060.130,-33.260,433.545,171.474,27.529,155.138
C02543=1060.136,-33.010,433.532,171.476,27.530,155.138
C02544=1060.142,-32.760,433.519,171.478,27.533,155.138
C02545=1060.149,-32.511,433.506,171.479,27.535,155.138
C02546=1060.154,-32.261,433.493,171.481,27.537,155.139
C02547=1060.161,-32.012,433.480,171.483,27.539,155.139
C02548=1060.167,-31.763,433.467,171.484,27.541,155.139
C02549=1060.173,-31.513,433.454,171.486,27.543,155.139
C02550=1060.180,-31.263,433.441,171.487,27.545,155.140
C02551=1060.186,-31.014,433.427,171.489,27.547,155.140
C02552=1060.191,-30.763,433.414,171.491,27.549,155.140
C02553=1060.197,-30.514,433.401,171.492,27.551,155.140
C02554=1060.203,-30.265,433.388,171.494,27.554,155.140
C02555=1060.209,-30.015,433.375,171.496,27.555,155.141
C02556=1060.216,-29.766,433.362,171.497,27.558,155.141
C02557=1060.222,-29.516,433.348,171.499,27.560,155.141
C02558=1060.229,-29.267,433.335,171.501,27.562,155.141
C02559=1060.235,-29.017,433.322,171.502,27.564,155.142
C02560=1060.241,-28.767,433.309,171.504,27.566,155.142
C02561=1060.247,-28.518,433.296,171.505,27.568,155.142
C02562=1060.253,-28.268,433.282,171.507,27.570,155.142
C02563=1060.259,-28.019,433.268,171.509,27.572,155.142
C02564=1060.265,-27.769,433.256,171.510,27.575,155.143
C02565=1060.271,-27.519,433.242,171.512,27.576,155.143
C02566=1060.278,-27.270,433.229,171.513,27.578,155.143
C02567=1060.284,-27.020,433.216,171.514,27.581,155.143
C02568=1060.291,-26.771,433.202,171.516,27.582,155.144
C02569=1060.296,-26.521,433.188,171.518,27.585,155.144
C02570=1060.302,-26.272,433.176,171.519,27.587,155.144
C02571=1060.308,-26.022,433.163,171.521,27.589,155.144
C02572=1060.314,-25.772,433.148,171.522,27.591,155.145
C02573=1060.320,-25.523,433.135,171.524,27.594,155.145
C02574=1060.327,-25.273,433.122,171.526,27.596,155.145
C02575=1060.332,-25.024,433.108,171.527,27.598,155.145
C02576=1060.338,-24.775,433.095,171.529,27.600,155.146
C02577=1060.345,-24.525,433.081,171.531,27.602,155.146
C02578=1060.351,-24.275,433.067,171.532,27.604,155.146
C02579=1060.357,-24.025,433.055,171.534,27.607,155.146
C02580=1060.363,-23.776,433.041,171.535,27.609,155.147
C02581=1060.368,-23.526,433.028,171.537,27.611,155.147
C02582=1060.375,-23.276,433.014,171.539,27.613,155.147
C02583=1060.381,-23.027,433.001,171.540,27.615,155.147
C02584=1060.387,-22.778,432.987,171.542,27.617,155.148
C02585=1060.393,-22.528,432.973,171.543,27.620,155.148
C02586=1060.400,-22.278,432.960,171.545,27.622,155.148
C02587=1060.405,-22.029,432.946,171.547,27.624,155.148
C02588=1060.412,-21.779,432.933,171.548,27.626,155.149
C02589=1060.418,-21.530,432.919,171.549,27.628,155.149
C02590=1060.424,-21.280,432.905,171.551,27.631,155.149
C02591=1060.430,-21.031,432.892,171.552,27.632,155.149
C02592=1060.436,-20.781,432.879,171.554,27.635,155.150
C02593=1060.442,-20.531,432.864,171.556,27.637,155.150
C02594=1060.449,-20.282,432.851,171.557,27.639,155.150
C02595=1060.454,-20.032,432.837,171.559,27.641,155.151
C02596=1060.460,-19.783,432.824,171.560,27.644,155.151
C02597=1060.467,-19.534,432.810,171.562,27.646,155.151
C02598=1060.473,-19.284,432.796,171.564,27.648,155.151
C02599=1060.479,-19.035,432.783,171.565,27.651,155.152
C02600=1060.486,-18.785,432.769,171.567,27.653,155.152
C02601=1060.492,-18.505,432.754,171.568,27.655,155.152
C02602=1060.499,-18.226,432.738,171.570,27.657,155.152
C02603=1060.506,-17.946,432.723,171.572,27.660,155.153
C02604=1060.513,-17.666,432.708,171.574,27.663,155.153
C02605=1060.519,-17.417,432.694,171.576,27.664,155.153
C02606=1060.525,-17.168,432.680,171.577,27.667,155.153
C02607=1060.531,-16.918,432.666,171.578,27.669,155.154
C02608=1060.538,-16.668,432.653,171.580,27.671,155.154
C02609=1060.543,-16.419,432.639,171.581,27.673,155.154
C02610=1060.550,-16.169,432.625,171.583,27.675,155.155
C02611=1060.556,-15.920,432.611,171.585,27.678,155.155
C02612=1060.563,-15.670,432.597,171.586,27.680,155.155
C02613=1060.569,-15.421,432.584,171.588,27.682,155.155
C02614=1060.574,-15.171,432.570,171.589,27.684,155.156
C02615=1060.581,-14.921,432.556,171.591,27.687,155.156
C02616=1060.587,-14.672,432.542,171.593,27.689,155.156
C02617=1060.592,-14.423,432.528,171.594,27.691,155.156
C02618=1060.599,-14.173,432.514,171.596,27.694,155.157
C02619=1060.605,-13.923,432.500,171.597,27.696,155.157
C02620=1060.610,-13.674,432.486,171.599,27.698,155.157
C02621=1060.617,-13.424,432.472,171.601,27.700,155.157
C02622=1060.623,-13.175,432.458,171.601,27.702,155.158
C02623=1060.629,-12.925,432.445,171.603,27.705,155.158
C02624=1060.635,-12.676,432.430,171.605,27.707,155.158
C02625=1060.641,-12.426,432.416,171.606,27.710,155.159
C02626=1060.648,-12.176,432.403,171.608,27.712,155.159
C02627=1060.653,-11.927,432.388,171.609,27.714,155.159
C02628=1060.659,-11.678,432.374,171.611,27.716,155.159
C02629=1060.666,-11.428,432.361,171.613,27.719,155.160
C02630=1060.671,-11.179,432.346,171.614,27.721,155.160
C02631=1060.678,-10.928,432.332,171.616,27.723,155.160
C02632=1060.684,-10.679,432.318,171.617,27.725,155.161
C02633=1060.690,-10.430,432.304,171.619,27.728,155.161
C02634=1060.696,-10.180,432.290,171.621,27.730,155.161
C02635=1060.702,-9.931,432.276,171.621,27.732,155.161
C02636=1060.708,-9.681,432.261,171.623,27.734,155.162
C02637=1060.714,-9.432,432.248,171.624,27.737,155.162
C02638=1060.721,-9.182,432.233,171.626,27.739,155.162
C02639=1060.726,-8.933,432.219,171.628,27.742,155.163
C02640=1060.732,-8.683,432.206,171.629,27.744,155.163
C02641=1060.739,-8.434,432.191,171.631,27.746,155.163
C02642=1060.744,-8.184,432.177,171.633,27.748,155.163
C02643=1060.751,-7.934,432.162,171.634,27.751,155.164
C02644=1060.757,-7.685,432.149,171.636,27.753,155.164
C02645=1060.763,-7.435,432.134,171.637,27.755,155.164
C02646=1060.769,-7.186,432.120,171.639,27.757,155.164
C02647=1060.776,-6.937,432.106,171.641,27.760,155.165
C02648=1060.781,-6.687,432.092,171.641,27.762,155.165
C02649=1060.788,-6.437,432.077,171.643,27.765,155.165
C02650=1060.794,-6.188,432.064,171.644,27.767,155.166
C02651=1060.800,-5.938,432.050,171.646,27.769,155.166
C02652=1060.806,-5.689,432.035,171.648,27.771,155.166
C02653=1060.813,-5.439,432.021,171.649,27.774,155.167
C02654=1060.818,-5.190,432.007,171.651,27.776,155.167
C02655=1060.825,-4.940,431.992,171.653,27.778,155.167
C02656=1060.830,-4.691,431.978,171.654,27.781,155.167
C02657=1060.837,-4.441,431.964,171.656,27.783,155.168
C02658=1060.843,-4.192,431.950,171.657,27.785,155.168
C02659=1060.849,-3.942,431.935,171.658,27.787,155.168
C02660=1060.855,-3.693,431.922,171.660,27.790,155.169
C02661=1060.862,-3.443,431.907,171.661,27.792,155.169
C02662=1060.868,-3.194,431.892,171.663,27.794,155.169
C02663=1060.874,-2.944,431.878,171.664,27.797,155.169
C02664=1060.880,-2.695,431.863,171.666,27.799,155.170
C02665=1060.887,-2.413,431.847,171.668,27.802,155.170
C02666=1060.893,-2.132,431.831,171.669,27.804,155.170
C02667=1060.900,-1.851,431.814,171.671,27.807,155.171
C02668=1060.907,-1.570,431.798,171.673,27.810,155.171
C02669=1060.913,-1.320,431.783,171.674,27.812,155.171
C02670=1060.919,-1.071,431.769,171.675,27.815,155.172
C02671=1060.925,-0.821,431.754,171.677,27.817,155.172
C02672=1060.931,-0.572,431.740,171.679,27.820,155.172
C02673=1060.937,-0.322,431.725,171.680,27.822,155.173
C02674=1060.943,-0.073,431.711,171.682,27.825,155.173
C02675=1060.949,0.177,431.696,171.683,27.827,155.173
C02676=1060.955,0.426,431.681,171.685,27.829,155.174
C02677=1060.961,0.676,431.667,171.687,27.832,155.174
C02678=1060.967,0.925,431.652,171.688,27.834,155.174
C02679=1060.973,1.175,431.638,171.689,27.836,155.175
C02680=1060.978,1.424,431.624,171.690,27.839,155.175
C02681=1060.985,1.674,431.609,171.692,27.841,155.175
C02682=1060.991,1.923,431.594,171.694,27.844,155.175
C02683=1060.997,2.173,431.579,171.695,27.846,155.176
C02684=1061.003,2.422,431.564,171.697,27.849,155.176
C02685=1061.009,2.672,431.550,171.698,27.851,155.176
C02686=1061.015,2.922,431.535,171.700,27.853,155.177
C02687=1061.021,3.170,431.521,171.702,27.856,155.177
C02688=1061.027,3.420,431.506,171.702,27.858,155.177
C02689=1061.034,3.670,431.491,171.704,27.860,155.178
C02690=1061.039,3.919,431.477,171.705,27.863,155.178
C02691=1061.046,4.169,431.462,171.707,27.865,155.178
C02692=1061.051,4.418,431.448,171.709,27.868,155.179
C02693=1061.058,4.668,431.433,171.710,27.870,155.179
C02694=1061.064,4.917,431.418,171.712,27.873,155.179
C02695=1061.070,5.166,431.403,171.713,27.875,155.179
C02696=1061.075,5.417,431.388,171.715,27.877,155.180
C02697=1061.081,5.666,431.374,171.716,27.880,155.180
C02698=1061.087,5.915,431.359,171.717,27.882,155.180
C02699=1061.094,6.165,431.344,171.719,27.884,155.181
C02700=1061.100,6.414,431.329,171.720,27.887,155.181
C02701=1061.106,6.664,431.314,171.722,27.889,155.181
C02702=1061.112,6.913,431.299,171.724,27.892,155.182
C02703=1061.118,7.162,431.285,171.725,27.894,155.182
C02704=1061.125,7.412,431.270,171.727,27.897,155.182
C02705=1061.131,7.662,431.255,171.728,27.899,155.183
C02706=1061.137,7.911,431.240,171.729,27.902,155.183
C02707=1061.143,8.160,431.225,171.731,27.904,155.183
C02708=1061.149,8.411,431.211,171.732,27.906,155.184
C02709=1061.155,8.659,431.197,171.734,27.909,155.184
C02710=1061.161,8.909,431.181,171.736,27.911,155.184
C02711=1061.167,9.159,431.166,171.737,27.913,155.184
C02712=1061.173,9.409,431.151,171.739,27.916,155.185
C02713=1061.179,9.658,431.137,171.740,27.918,155.185
C02714=1061.186,9.907,431.122,171.741,27.920,155.185
C02715=1061.192,10.157,431.107,171.743,27.923,155.186
C02716=1061.198,10.406,431.092,171.744,27.925,155.186
C02717=1061.204,10.656,431.077,171.746,27.928,155.186
C02718=1061.211,10.905,431.061,171.747,27.931,155.187
C02719=1061.217,11.154,431.046,171.749,27.933,155.187
C02720=1061.222,11.404,431.031,171.751,27.935,155.187
C02721=1061.229,11.653,431.016,171.752,27.938,155.188
C02722=1061.235,11.903,431.001,171.753,27.940,155.188
C02723=1061.241,12.153,430.986,171.754,27.942,155.188
C02724=1061.247,12.402,430.972,171.756,27.945,155.189
C02725=1061.254,12.651,430.957,171.758,27.947,155.189
C02726=1061.260,12.901,430.942,171.759,27.949,155.189
C02727=1061.266,13.150,430.927,171.761,27.952,155.190
C02728=1061.272,13.399,430.912,171.762,27.954,155.190
C02729=1061.279,13.683,430.895,171.764,27.957,155.190
C02730=1061.286,13.965,430.878,171.766,27.960,155.191
C02731=1061.292,14.249,430.861,171.767,27.962,155.191
C02732=1061.300,14.532,430.844,171.769,27.965,155.191
C02733=1061.306,14.782,430.829,171.770,27.968,155.192
C02734=1061.312,15.031,430.813,171.772,27.970,155.192
C02735=1061.319,15.281,430.798,171.773,27.973,155.192
C02736=1061.324,15.530,430.783,171.775,27.975,155.193
C02737=1061.330,15.780,430.767,171.777,27.978,155.193
C02738=1061.336,16.029,430.753,171.777,27.980,155.193
C02739=1061.343,16.278,430.737,171.779,27.982,155.194
C02740=1061.348,16.528,430.722,171.781,27.985,155.194
C02741=1061.354,16.777,430.707,171.782,27.987,155.194
C02742=1061.361,17.027,430.692,171.784,27.990,155.195
C02743=1061.367,17.276,430.676,171.785,27.993,155.195
C02744=1061.373,17.526,430.661,171.787,27.995,155.195
C02745=1061.378,17.775,430.645,171.788,27.997,155.196
C02746=1061.385,18.025,430.630,171.789,28.000,155.196
C02747=1061.391,18.274,430.615,171.791,28.002,155.196
C02748=1061.397,18.524,430.599,171.792,28.005,155.197
C02749=1061.403,18.774,430.584,171.794,28.007,155.197
C02750=1061.409,19.022,430.569,171.795,28.010,155.197
C02751=1061.415,19.272,430.553,171.797,28.012,155.198
C02752=1061.421,19.522,430.539,171.799,28.015,155.198
C02753=1061.427,19.771,430.523,171.799,28.017,155.198
C02754=1061.434,20.021,430.507,171.801,28.020,155.199
C02755=1061.440,20.270,430.492,171.803,28.022,155.199
C02756=1061.445,20.519,430.476,171.804,28.025,155.199
C02757=1061.452,20.768,430.462,171.806,28.027,155.200
C02758=1061.458,21.018,430.446,171.807,28.030,155.200
C02759=1061.464,21.267,430.430,171.809,28.032,155.200
C02760=1061.470,21.517,430.415,171.810,28.035,155.201
C02761=1061.476,21.767,430.400,171.811,28.037,155.201
C02762=1061.482,22.016,430.384,171.813,28.040,155.201
C02763=1061.488,22.265,430.369,171.814,28.042,155.202
C02764=1061.494,22.515,430.353,171.816,28.045,155.202
C02765=1061.500,22.764,430.338,171.818,28.047,155.202
C02766=1061.506,23.014,430.322,171.819,28.050,155.203
C02767=1061.513,23.263,430.307,171.820,28.052,155.203
C02768=1061.518,23.513,430.291,171.821,28.055,155.203
C02769=1061.524,23.762,430.276,171.823,28.057,155.204
C02770=1061.530,24.012,430.260,171.825,28.060,155.204
C02771=1061.537,24.261,430.245,171.826,28.062,155.204
C02772=1061.542,24.511,430.229,171.828,28.065,155.205
C02773=1061.549,24.760,430.213,171.829,28.068,155.205
C02774=1061.555,25.010,430.198,171.830,28.070,155.205
C02775=1061.561,25.259,430.182,171.832,28.073,155.206
C02776=1061.567,25.509,430.167,171.833,28.075,155.206
C02777=1061.572,25.757,430.151,171.835,28.078,155.206
C02778=1061.579,26.007,430.136,171.836,28.080,155.207
C02779=1061.585,26.256,430.120,171.838,28.083,155.207
C02780=1061.591,26.506,430.105,171.839,28.085,155.207
C02781=1061.597,26.755,430.088,171.840,28.088,155.208
C02782=1061.604,27.004,430.073,171.842,28.090,155.208
C02783=1061.609,27.254,430.057,171.843,28.093,155.208
C02784=1061.615,27.504,430.041,171.845,28.095,155.209
C02785=1061.622,27.753,430.026,171.847,28.098,155.209
C02786=1061.628,28.003,430.010,171.848,28.101,155.210
C02787=1061.634,28.252,429.995,171.849,28.103,155.210
C02788=1061.640,28.502,429.978,171.850,28.105,155.210
C02789=1061.646,28.751,429.962,171.852,28.108,155.211
C02790=1061.652,29.001,429.947,171.854,28.110,155.211
C02791=1061.658,29.249,429.931,171.855,28.113,155.211
C02792=1061.664,29.499,429.915,171.857,28.115,155.212
C02793=1061.671,29.784,429.897,171.858,28.118,155.212
C02794=1061.678,30.068,429.879,171.860,28.121,155.212
C02795=1061.685,30.353,429.862,171.861,28.124,155.213
C02796=1061.691,30.637,429.843,171.863,28.127,155.213
C02797=1061.697,30.886,429.828,171.865,28.129,155.214
C02798=1061.703,31.136,429.812,171.866,28.132,155.214
C02799=1061.709,31.385,429.795,171.868,28.135,155.214
C02800=1061.715,31.635,429.779,171.868,28.137,155.215
C02801=1061.722,31.884,429.764,171.870,28.140,155.215
C02802=1061.728,32.134,429.748,171.872,28.142,155.215
C02803=1061.734,32.383,429.732,171.873,28.145,155.216
C02804=1061.739,32.633,429.716,171.875,28.148,155.216
C02805=1061.745,32.882,429.700,171.876,28.150,155.216
C02806=1061.752,33.131,429.684,171.878,28.153,155.217
C02807=1061.758,33.381,429.668,171.879,28.155,155.217
C02808=1061.764,33.631,429.652,171.880,28.158,155.217
C02809=1061.769,33.880,429.636,171.882,28.160,155.218
C02810=1061.776,34.129,429.621,171.883,28.163,155.218
C02811=1061.782,34.378,429.604,171.885,28.165,155.219
C02812=1061.788,34.628,429.588,171.887,28.168,155.219
C02813=1061.794,34.878,429.572,171.887,28.170,155.219
C02814=1061.800,35.127,429.557,171.889,28.173,155.220
C02815=1061.806,35.376,429.541,171.890,28.175,155.220
C02816=1061.812,35.625,429.524,171.892,28.178,155.220
C02817=1061.818,35.875,429.508,171.894,28.181,155.221
C02818=1061.824,36.124,429.492,171.895,28.183,155.221
C02819=1061.831,36.373,429.476,171.897,28.186,155.221
C02820=1061.837,36.623,429.461,171.897,28.188,155.222
C02821=1061.842,36.872,429.444,171.899,28.191,155.222
C02822=1061.848,37.122,429.428,171.901,28.194,155.222
C02823=1061.854,37.371,429.412,171.902,28.196,155.223
C02824=1061.862,37.621,429.396,171.904,28.199,155.223
C02825=1061.868,37.870,429.380,171.905,28.201,155.223
C02826=1061.874,38.120,429.363,171.906,28.203,155.224
C02827=1061.880,38.369,429.347,171.908,28.206,155.224
C02828=1061.885,38.618,429.331,171.909,28.209,155.225
C02829=1061.891,38.868,429.315,171.911,28.211,155.225
C02830=1061.897,39.117,429.298,171.912,28.214,155.225
C02831=1061.903,39.366,429.282,171.914,28.217,155.226
C02832=1061.909,39.616,429.266,171.915,28.219,155.226
C02833=1061.915,39.866,429.250,171.916,28.222,155.226
C02834=1061.921,40.115,429.234,171.918,28.224,155.227
C02835=1061.927,40.364,429.218,171.919,28.227,155.227
C02836=1061.933,40.614,429.201,171.921,28.229,155.227
C02837=1061.939,40.863,429.185,171.923,28.232,155.228
C02838=1061.945,41.112,429.169,171.923,28.235,155.228
C02839=1061.951,41.361,429.152,171.925,28.238,155.229
C02840=1061.957,41.610,429.136,171.926,28.240,155.229
C02841=1061.963,41.860,429.119,171.928,28.243,155.229
C02842=1061.969,42.110,429.103,171.930,28.245,155.230
C02843=1061.975,42.359,429.087,171.931,28.248,155.230
C02844=1061.981,42.609,429.070,171.933,28.250,155.230
C02845=1061.987,42.858,429.054,171.933,28.253,155.231
C02846=1061.993,43.107,429.038,171.935,28.255,155.231
C02847=1061.999,43.357,429.022,171.937,28.258,155.231
C02848=1062.005,43.606,429.005,171.938,28.261,155.232
C02849=1062.010,43.856,428.988,171.940,28.264,155.232
C02850=1062.017,44.106,428.972,171.941,28.266,155.233
C02851=1062.023,44.355,428.956,171.942,28.268,155.233
C02852=1062.029,44.604,428.939,171.944,28.271,155.233
C02853=1062.035,44.853,428.922,171.945,28.274,155.234
C02854=1062.040,45.103,428.905,171.947,28.277,155.234
C02855=1062.046,45.352,428.889,171.948,28.279,155.234
C02856=1062.052,45.601,428.873,171.950,28.282,155.235
C02857=1062.059,45.886,428.854,171.952,28.285,155.235
C02858=1062.066,46.170,428.835,171.953,28.288,155.236
C02859=1062.073,46.454,428.816,171.955,28.291,155.236
C02860=1062.080,46.739,428.797,171.956,28.294,155.237
C02861=1062.085,46.989,428.780,171.958,28.297,155.237
C02862=1062.091,47.238,428.764,171.959,28.299,155.237
C02863=1062.097,47.487,428.748,171.960,28.302,155.238
C02864=1062.102,47.736,428.730,171.962,28.305,155.238
C02865=1062.108,47.986,428.714,171.963,28.307,155.238
C02866=1062.115,48.236,428.697,171.965,28.310,155.239
C02867=1062.121,48.485,428.681,171.966,28.312,155.239
C02868=1062.126,48.734,428.663,171.968,28.315,155.240
C02869=1062.132,48.983,428.647,171.969,28.318,155.240
C02870=1062.138,49.233,428.631,171.970,28.320,155.240
C02871=1062.144,49.482,428.614,171.972,28.323,155.241
C02872=1062.150,49.732,428.597,171.973,28.325,155.241
C02873=1062.156,49.981,428.580,171.975,28.328,155.241
C02874=1062.162,50.230,428.563,171.977,28.331,155.242
C02875=1062.168,50.479,428.547,171.977,28.334,155.242
C02876=1062.174,50.729,428.530,171.979,28.336,155.243
C02877=1062.180,50.978,428.513,171.980,28.339,155.243
C02878=1062.186,51.228,428.497,171.982,28.341,155.243
C02879=1062.192,51.477,428.480,171.984,28.344,155.244
C02880=1062.198,51.726,428.463,171.985,28.347,155.244
C02881=1062.204,51.976,428.447,171.986,28.349,155.244
C02882=1062.210,52.226,428.429,171.987,28.352,155.245
C02883=1062.216,52.475,428.412,171.989,28.355,155.245
C02884=1062.222,52.724,428.396,171.991,28.357,155.246
C02885=1062.228,52.973,428.379,171.992,28.360,155.246
C02886=1062.233,53.222,428.362,171.994,28.362,155.246
C02887=1062.240,53.472,428.346,171.995,28.365,155.247
C02888=1062.246,53.721,428.329,171.996,28.368,155.247
C02889=1062.251,53.971,428.312,171.998,28.371,155.247
C02890=1062.258,54.220,428.295,171.999,28.373,155.248
C02891=1062.264,54.470,428.278,172.001,28.376,155.248
C02892=1062.270,54.719,428.261,172.002,28.378,155.249
C02893=1062.276,54.968,428.245,172.003,28.381,155.249
C02894=1062.282,55.217,428.227,172.005,28.383,155.249
C02895=1062.288,55.467,428.210,172.006,28.386,155.250
C02896=1062.294,55.716,428.193,172.008,28.389,155.250
C02897=1062.300,55.965,428.177,172.010,28.391,155.250
C02898=1062.306,56.215,428.159,172.011,28.394,155.251
C02899=1062.312,56.464,428.143,172.012,28.396,155.251
C02900=1062.318,56.713,428.126,172.013,28.399,155.252
C02901=1062.324,56.963,428.109,172.015,28.402,155.252
C02902=1062.330,57.212,428.092,172.017,28.405,155.252
C02903=1062.336,57.461,428.076,172.018,28.407,155.253
C02904=1062.342,57.711,428.058,172.020,28.410,155.253
C02905=1062.348,57.960,428.041,172.020,28.412,155.253
C02906=1062.354,58.210,428.024,172.022,28.415,155.254
C02907=1062.360,58.460,428.007,172.024,28.417,155.254
C02908=1062.367,58.708,427.990,172.025,28.420,155.255
C02909=1062.372,58.957,427.973,172.027,28.423,155.255
C02910=1062.379,59.207,427.956,172.029,28.425,155.255
C02911=1062.385,59.456,427.939,172.029,28.427,155.256
C02912=1062.390,59.706,427.922,172.031,28.430,155.256
C02913=1062.397,59.955,427.905,172.032,28.433,155.256
C02914=1062.403,60.204,427.888,172.034,28.435,155.257
C02915=1062.409,60.454,427.871,172.036,28.438,155.257
C02916=1062.415,60.703,427.854,172.037,28.441,155.257
C02917=1062.421,60.952,427.836,172.039,28.444,155.258
C02918=1062.427,61.202,427.819,172.040,28.446,155.258
C02919=1062.434,61.451,427.802,172.041,28.448,155.259
C02920=1062.440,61.701,427.785,172.043,28.451,155.259
C02921=1062.446,61.985,427.766,172.044,28.454,155.259
C02922=1062.454,62.269,427.746,172.046,28.457,155.260
C02923=1062.461,62.553,427.727,172.047,28.460,155.260
C02924=1062.467,62.837,427.707,172.049,28.463,155.261
C02925=1062.474,63.086,427.690,172.051,28.465,155.261
C02926=1062.480,63.336,427.673,172.052,28.468,155.261
C02927=1062.486,63.585,427.655,172.054,28.471,155.262
C02928=1062.492,63.834,427.638,172.055,28.473,155.262
C02929=1062.498,64.083,427.621,172.057,28.476,155.262
C02930=1062.505,64.334,427.604,172.059,28.478,155.263
C02931=1062.510,64.583,427.586,172.059,28.481,155.263
C02932=1062.516,64.831,427.569,172.061,28.484,155.264
C02933=1062.522,65.081,427.551,172.062,28.487,155.264
C02934=1062.528,65.331,427.535,172.064,28.489,155.264
C02935=1062.534,65.580,427.517,172.066,28.492,155.265
C02936=1062.540,65.829,427.500,172.067,28.494,155.265
C02937=1062.546,66.078,427.482,172.068,28.497,155.266
C02938=1062.552,66.328,427.465,172.070,28.500,155.266
C02939=1062.558,66.577,427.447,172.071,28.502,155.266
C02940=1062.564,66.827,427.431,172.073,28.505,155.267
C02941=1062.570,67.076,427.413,172.074,28.507,155.267
C02942=1062.576,67.326,427.395,172.076,28.510,155.267
C02943=1062.582,67.574,427.378,172.078,28.513,155.268
C02944=1062.588,67.824,427.360,172.078,28.516,155.268
C02945=1062.594,68.073,427.343,172.080,28.518,155.269
C02946=1062.599,68.322,427.325,172.082,28.520,155.269
C02947=1062.606,68.572,427.308,172.083,28.523,155.269
C02948=1062.612,68.821,427.290,172.085,28.526,155.270
C02949=1062.618,69.070,427.272,172.086,28.529,155.270
C02950=1062.624,69.320,427.256,172.087,28.531,155.271
C02951=1062.630,69.569,427.238,172.089,28.534,155.271
C02952=1062.636,69.818,427.220,172.090,28.536,155.271
C02953=1062.642,70.068,427.202,172.092,28.539,155.272
C02954=1062.648,70.317,427.186,172.093,28.542,155.272
C02955=1062.654,70.567,427.168,172.095,28.545,155.272
C02956=1062.660,70.816,427.150,172.096,28.547,155.273
C02957=1062.665,71.065,427.132,172.097,28.550,155.273
C02958=1062.671,71.314,427.115,172.099,28.553,155.274
C02959=1062.677,71.563,427.098,172.101,28.555,155.274
C02960=1062.684,71.813,427.080,172.102,28.558,155.274
C02961=1062.689,72.062,427.062,172.104,28.561,155.275
C02962=1062.695,72.312,427.044,172.105,28.563,155.275
C02963=1062.701,72.561,427.027,172.106,28.566,155.276
C02964=1062.707,72.810,427.009,172.108,28.569,155.276
C02965=1062.713,73.059,426.991,172.109,28.571,155.276
C02966=1062.720,73.308,426.973,172.111,28.574,155.277
C02967=1062.725,73.557,426.955,172.112,28.576,155.277
C02968=1062.731,73.807,426.938,172.114,28.579,155.277
C02969=1062.737,74.056,426.920,172.115,28.582,155.278
C02970=1062.743,74.306,426.902,172.116,28.584,155.278
C02971=1062.748,74.555,426.884,172.118,28.587,155.279
C02972=1062.755,74.804,426.867,172.120,28.590,155.279
C02973=1062.761,75.053,426.850,172.121,28.593,155.279
C02974=1062.767,75.303,426.832,172.123,28.595,155.280
C02975=1062.773,75.552,426.813,172.124,28.598,155.280
C02976=1062.779,75.801,426.795,172.125,28.600,155.281
C02977=1062.785,76.051,426.777,172.127,28.603,155.281
C02978=1062.790,76.300,426.760,172.128,28.606,155.281
C02979=1062.797,76.550,426.742,172.130,28.609,155.282
C02980=1062.802,76.799,426.724,172.131,28.611,155.282
C02981=1062.809,77.048,426.706,172.133,28.614,155.282
C02982=1062.815,77.297,426.689,172.135,28.616,155.283
C02983=1062.821,77.546,426.671,172.135,28.619,155.283
C02984=1062.827,77.796,426.653,172.137,28.622,155.284
C02985=1062.833,78.079,426.632,172.139,28.624,155.284
C02986=1062.840,78.364,426.612,172.140,28.628,155.285
C02987=1062.847,78.648,426.591,172.143,28.631,155.285
C02988=1062.853,78.932,426.571,172.144,28.634,155.285
C02989=1062.859,79.182,426.553,172.146,28.637,155.286
C02990=1062.866,79.431,426.534,172.146,28.639,155.286
C02991=1062.871,79.680,426.517,172.148,28.642,155.287
C02992=1062.877,79.930,426.499,172.150,28.644,155.287
C02993=1062.883,80.178,426.481,172.151,28.647,155.287
C02994=1062.889,80.428,426.463,172.153,28.650,155.288
C02995=1062.895,80.677,426.445,172.155,28.653,155.288
C02996=1062.901,80.926,426.426,172.156,28.655,155.289
C02997=1062.907,81.176,426.408,172.157,28.658,155.289
C02998=1062.912,81.425,426.390,172.158,28.661,155.289
C02999=1062.919,81.674,426.372,172.160,28.664,155.290
C03000=1062.924,81.923,426.354,172.162,28.666,155.290
C03001=1062.930,82.173,426.336,172.163,28.669,155.291
C03002=1062.936,82.421,426.318,172.165,28.672,155.291
C03003=1062.942,82.671,426.300,172.166,28.674,155.291
C03004=1062.949,82.920,426.281,172.167,28.677,155.292
C03005=1062.953,83.169,426.263,172.169,28.680,155.292
C03006=1062.959,83.419,426.245,172.170,28.682,155.292
C03007=1062.966,83.668,426.227,172.172,28.685,155.293
C03008=1062.971,83.917,426.209,172.174,28.688,155.293
C03009=1062.978,84.167,426.190,172.175,28.690,155.294
C03010=1062.984,84.416,426.172,172.177,28.693,155.294
C03011=1062.989,84.665,426.154,172.178,28.696,155.295
C03012=1062.995,84.915,426.136,172.179,28.699,155.295
C03013=1063.001,85.164,426.118,172.181,28.701,155.295
C03014=1063.007,85.413,426.099,172.182,28.704,155.296
C03015=1063.013,85.663,426.082,172.184,28.707,155.296
C03016=1063.019,85.911,426.063,172.186,28.709,155.296
C03017=1063.024,86.161,426.045,172.187,28.712,155.297
C03018=1063.031,86.410,426.026,172.188,28.714,155.297
C03019=1063.037,86.660,426.008,172.190,28.717,155.298
C03020=1063.043,86.908,425.990,172.191,28.720,155.298
C03021=1063.049,87.158,425.972,172.193,28.723,155.298
C03022=1063.055,87.407,425.953,172.194,28.725,155.299
C03023=1063.060,87.656,425.934,172.196,28.728,155.299
C03024=1063.067,87.906,425.916,172.198,28.731,155.300
C03025=1063.073,88.155,425.898,172.199,28.733,155.300
C03026=1063.078,88.404,425.880,172.200,28.736,155.300
C03027=1063.085,88.653,425.862,172.202,28.738,155.301
C03028=1063.090,88.903,425.843,172.203,28.741,155.301
C03029=1063.097,89.152,425.824,172.205,28.744,155.302
C03030=1063.103,89.401,425.806,172.206,28.747,155.302
C03031=1063.109,89.650,425.788,172.208,28.749,155.302
C03032=1063.115,89.899,425.770,172.210,28.752,155.303
C03033=1063.120,90.150,425.751,172.211,28.754,155.303
C03034=1063.126,90.398,425.733,172.212,28.757,155.303
C03035=1063.133,90.647,425.714,172.214,28.760,155.304
C03036=1063.139,90.897,425.696,172.215,28.762,155.304
C03037=1063.145,91.146,425.677,172.217,28.765,155.305
C03038=1063.150,91.395,425.659,172.218,28.768,155.305
C03039=1063.156,91.645,425.640,172.220,28.771,155.305
C03040=1063.162,91.894,425.621,172.222,28.773,155.306
C03041=1063.168,92.142,425.603,172.223,28.776,155.306
C03042=1063.174,92.392,425.584,172.224,28.779,155.307
C03043=1063.180,92.641,425.566,172.226,28.781,155.307
C03044=1063.185,92.891,425.547,172.227,28.784,155.307
C03045=1063.191,93.139,425.528,172.229,28.787,155.308
C03046=1063.197,93.389,425.509,172.230,28.790,155.308
C03047=1063.203,93.638,425.491,172.232,28.793,155.309
C03048=1063.209,93.888,425.472,172.234,28.795,155.309
C03049=1063.216,94.172,425.451,172.235,28.798,155.309
C03050=1063.223,94.456,425.430,172.237,28.801,155.310
C03051=1063.229,94.740,425.408,172.238,28.804,155.310
C03052=1063.236,95.024,425.387,172.240,28.807,155.311
C03053=1063.241,95.273,425.369,172.242,28.810,155.311
C03054=1063.247,95.522,425.350,172.243,28.812,155.312
C03055=1063.253,95.771,425.331,172.245,28.815,155.312
C03056=1063.260,96.020,425.312,172.247,28.818,155.312
C03057=1063.266,96.270,425.294,172.248,28.821,155.313
C03058=1063.271,96.519,425.275,172.250,28.823,155.313
C03059=1063.277,96.768,425.257,172.251,28.826,155.314
C03060=1063.283,97.017,425.237,172.252,28.829,155.314
C03061=1063.289,97.267,425.219,172.254,28.831,155.314
C03062=1063.295,97.516,425.199,172.255,28.834,155.315
C03063=1063.301,97.764,425.181,172.257,28.837,155.315
C03064=1063.307,98.014,425.162,172.259,28.840,155.316
C03065=1063.313,98.263,425.143,172.260,28.842,155.316
C03066=1063.318,98.513,425.125,172.262,28.845,155.316
C03067=1063.325,98.762,425.106,172.264,28.847,155.317
C03068=1063.330,99.012,425.087,172.265,28.850,155.317
C03069=1063.337,99.261,425.068,172.266,28.853,155.318
C03070=1063.342,99.509,425.049,172.267,28.855,155.318
C03071=1063.348,99.759,425.031,172.269,28.858,155.318
C03072=1063.354,100.008,425.011,172.271,28.861,155.319
C03073=1063.361,100.257,424.993,172.272,28.864,155.319
C03074=1063.366,100.507,424.973,172.274,28.866,155.320
C03075=1063.373,100.756,424.955,172.276,28.869,155.320
C03076=1063.378,101.005,424.936,172.277,28.871,155.320
C03077=1063.384,101.255,424.916,172.279,28.874,155.321
C03078=1063.390,101.503,424.898,172.281,28.877,155.321
C03079=1063.396,101.752,424.879,172.281,28.879,155.322
C03080=1063.401,102.002,424.860,172.283,28.882,155.322
C03081=1063.407,102.251,424.840,172.285,28.885,155.322
C03082=1063.413,102.500,424.822,172.286,28.888,155.323
C03083=1063.419,102.750,424.802,172.288,28.890,155.323
C03084=1063.425,102.999,424.782,172.289,28.893,155.324
C03085=1063.431,103.247,424.764,172.291,28.896,155.324
C03086=1063.437,103.497,424.745,172.293,28.899,155.324
C03087=1063.442,103.746,424.726,172.294,28.901,155.325
C03088=1063.448,103.995,424.706,172.296,28.904,155.325
C03089=1063.454,104.245,424.688,172.297,28.907,155.326
C03090=1063.460,104.494,424.669,172.298,28.909,155.326
C03091=1063.466,104.743,424.649,172.300,28.912,155.326
C03092=1063.471,104.993,424.630,172.301,28.915,155.327
C03093=1063.478,105.241,424.611,172.303,28.918,155.327
C03094=1063.483,105.490,424.592,172.305,28.920,155.328
C03095=1063.489,105.739,424.573,172.306,28.923,155.328
C03096=1063.495,105.989,424.553,172.308,28.926,155.328
C03097=1063.501,106.238,424.535,172.310,28.929,155.329
C03098=1063.507,106.487,424.515,172.311,28.931,155.329
C03099=1063.513,106.736,424.496,172.313,28.934,155.330
C03100=1063.518,106.986,424.476,172.315,28.937,155.330
C03101=1063.525,107.235,424.458,172.315,28.939,155.330
C03102=1063.530,107.484,424.438,172.317,28.942,155.331
C03103=1063.536,107.733,424.418,172.318,28.945,155.331
C03104=1063.542,107.983,424.399,172.320,28.948,155.332
C03105=1063.548,108.232,424.380,172.322,28.950,155.332
C03106=1063.554,108.481,424.361,172.323,28.953,155.332
C03107=1063.560,108.730,424.341,172.325,28.956,155.333
C03108=1063.566,108.979,424.322,172.327,28.959,155.333
C03109=1063.572,109.229,424.303,172.328,28.961,155.334
C03110=1063.578,109.478,424.283,172.330,28.964,155.334
C03111=1063.584,109.727,424.264,172.332,28.966,155.334
C03112=1063.590,109.976,424.245,172.333,28.969,155.335
C03113=1063.596,110.260,424.223,172.335,28.972,155.335
C03114=1063.603,110.544,424.201,172.336,28.975,155.336
C03115=1063.610,110.828,424.178,172.338,28.978,155.336
C03116=1063.617,111.112,424.157,172.340,28.981,155.337
C03117=1063.623,111.335,424.139,172.341,28.984,155.337
C03118=1063.628,111.558,424.122,172.343,28.986,155.337
C03119=1063.633,111.808,424.102,172.345,28.989,155.338
C03120=1063.639,112.057,424.083,172.346,28.992,155.338
C03121=1063.645,112.306,424.063,172.348,28.994,155.338
C03122=1063.651,112.555,424.044,172.350,28.997,155.339
C03123=1063.657,112.804,424.024,172.351,29.000,155.339
C03124=1063.662,113.054,424.005,172.353,29.002,155.340
C03125=1063.668,113.303,423.985,172.354,29.005,155.340
C03126=1063.674,113.552,423.966,172.355,29.008,155.341
C03127=1063.680,113.801,423.946,172.357,29.010,155.341
C03128=1063.686,114.050,423.926,172.358,29.013,155.341
C03129=1063.691,114.300,423.907,172.360,29.016,155.342
C03130=1063.697,114.548,423.887,172.362,29.019,155.342
C03131=1063.703,114.798,423.868,172.363,29.021,155.343
C03132=1063.709,115.047,423.848,172.365,29.024,155.343
C03133=1063.714,115.296,423.828,172.367,29.027,155.343
C03134=1063.720,115.545,423.808,172.368,29.030,155.344
C03135=1063.726,115.794,423.788,172.370,29.032,155.344
C03136=1063.732,116.043,423.769,172.372,29.035,155.345
C03137=1063.738,116.292,423.749,172.373,29.038,155.345
C03138=1063.743,116.542,423.730,172.375,29.041,155.346
C03139=1063.749,116.791,423.709,172.376,29.044,155.346
C03140=1063.754,117.040,423.690,172.378,29.047,155.346
C03141=1063.760,117.289,423.670,172.380,29.049,155.347
C03142=1063.767,117.539,423.650,172.381,29.052,155.347
C03143=1063.773,117.788,423.630,172.382,29.055,155.348
C03144=1063.779,118.037,423.611,172.384,29.057,155.348
C03145=1063.783,118.287,423.591,172.385,29.060,155.348
C03146=1063.789,118.535,423.571,172.387,29.063,155.349
C03147=1063.795,118.784,423.551,172.389,29.066,155.349
C03148=1063.801,119.034,423.532,172.390,29.068,155.350
C03149=1063.807,119.282,423.512,172.392,29.071,155.350
C03150=1063.812,119.532,423.491,172.394,29.074,155.350
C03151=1063.818,119.781,423.472,172.395,29.077,155.351
C03152=1063.824,120.030,423.452,172.397,29.079,155.351
C03153=1063.830,120.279,423.432,172.398,29.082,155.352
C03154=1063.835,120.528,423.412,172.400,29.085,155.352
C03155=1063.842,120.778,423.392,172.402,29.087,155.352
C03156=1063.848,121.027,423.372,172.403,29.090,155.353
C03157=1063.854,121.276,423.352,172.405,29.093,155.353
C03158=1063.859,121.525,423.333,172.407,29.096,155.354
C03159=1063.865,121.774,423.312,172.408,29.098,155.354
C03160=1063.871,122.023,423.292,172.410,29.101,155.354
C03161=1063.877,122.272,423.272,172.412,29.104,155.355
C03162=1063.882,122.521,423.253,172.413,29.107,155.355
C03163=1063.888,122.771,423.232,172.415,29.110,155.356
C03164=1063.894,123.020,423.212,172.417,29.113,155.356
C03165=1063.900,123.269,423.192,172.418,29.115,155.357
C03166=1063.906,123.518,423.173,172.420,29.118,155.357
C03167=1063.911,123.767,423.152,172.421,29.121,155.357
C03168=1063.917,124.016,423.132,172.423,29.124,155.358
C03169=1063.924,124.266,423.112,172.425,29.126,155.358
C03170=1063.930,124.514,423.092,172.427,29.128,155.359
C03171=1063.935,124.763,423.071,172.428,29.131,155.359
C03172=1063.941,125.013,423.052,172.430,29.134,155.359
C03173=1063.947,125.262,423.032,172.431,29.137,155.360
C03174=1063.953,125.511,423.012,172.433,29.139,155.360
C03175=1063.963,125.932,422.978,172.436,29.144,155.361
C03176=1063.972,126.353,422.944,172.438,29.149,155.362
C03177=1063.983,126.775,422.910,172.441,29.154,155.362
C03178=1063.992,127.196,422.876,172.444,29.158,155.363
C03179=1063.998,127.446,422.855,172.445,29.160,155.363
C03180=1064.004,127.695,422.835,172.447,29.163,155.364
C03181=1064.010,127.944,422.815,172.449,29.166,155.364
C03182=1064.016,128.193,422.795,172.450,29.169,155.365
C03183=1064.022,128.443,422.774,172.452,29.171,155.365
C03184=1064.028,128.691,422.754,172.454,29.174,155.365
C03185=1064.034,128.940,422.734,172.455,29.177,155.366
C03186=1064.039,129.189,422.714,172.457,29.179,155.366
C03187=1064.046,129.439,422.693,172.459,29.182,155.367
C03188=1064.052,129.688,422.673,172.460,29.185,155.367
C03189=1064.057,129.937,422.653,172.462,29.188,155.367
C03190=1064.064,130.186,422.632,172.464,29.190,155.368
C03191=1064.070,130.435,422.612,172.465,29.193,155.368
C03192=1064.075,130.684,422.592,172.467,29.196,155.369
C03193=1064.082,130.934,422.572,172.469,29.198,155.369
C03194=1064.088,131.183,422.552,172.470,29.201,155.369
C03195=1064.093,131.432,422.531,172.472,29.203,155.370
C03196=1064.100,131.681,422.511,172.474,29.206,155.370
C03197=1064.106,131.930,422.491,172.475,29.209,155.370
C03198=1064.111,132.179,422.469,172.477,29.212,155.371
C03199=1064.117,132.427,422.449,172.479,29.214,155.371
C03200=1064.123,132.677,422.429,172.480,29.217,155.372
C03201=1064.128,132.926,422.408,172.482,29.220,155.372
C03202=1064.134,133.175,422.388,172.484,29.223,155.373
C03203=1064.140,133.425,422.367,172.486,29.226,155.373
C03204=1064.146,133.673,422.346,172.488,29.229,155.373
C03205=1064.152,133.922,422.326,172.489,29.231,155.374
C03206=1064.158,134.171,422.306,172.491,29.234,155.374
C03207=1064.163,134.421,422.285,172.493,29.237,155.375
C03208=1064.169,134.670,422.264,172.494,29.240,155.375
C03209=1064.175,134.918,422.244,172.496,29.242,155.375
C03210=1064.181,135.168,422.223,172.498,29.245,155.376
C03211=1064.187,135.417,422.203,172.499,29.248,155.376
C03212=1064.192,135.666,422.182,172.501,29.250,155.377
C03213=1064.198,135.915,422.161,172.503,29.253,155.377
C03214=1064.204,136.164,422.141,172.504,29.256,155.377
C03215=1064.210,136.413,422.120,172.506,29.259,155.378
C03216=1064.216,136.663,422.100,172.508,29.261,155.378
C03217=1064.222,136.911,422.079,172.509,29.264,155.379
C03218=1064.228,137.161,422.058,172.511,29.267,155.379
C03219=1064.234,137.410,422.038,172.513,29.269,155.380
C03220=1064.239,137.658,422.016,172.514,29.272,155.380
C03221=1064.245,137.908,421.996,172.516,29.275,155.380
C03222=1064.251,138.157,421.976,172.518,29.278,155.381
C03223=1064.257,138.405,421.954,172.519,29.280,155.381
C03224=1064.262,138.655,421.933,172.521,29.283,155.382
C03225=1064.268,138.904,421.913,172.523,29.286,155.382
C03226=1064.275,139.153,421.892,172.524,29.289,155.383
C03227=1064.280,139.402,421.871,172.527,29.292,155.383
C03228=1064.286,139.651,421.851,172.529,29.295,155.383
C03229=1064.292,139.900,421.830,172.530,29.297,155.384
C03230=1064.297,140.150,421.809,172.532,29.300,155.384
C03231=1064.303,140.399,421.787,172.534,29.303,155.385
C03232=1064.309,140.648,421.768,172.535,29.306,155.385
C03233=1064.315,140.896,421.746,172.537,29.308,155.385
C03234=1064.321,141.146,421.725,172.539,29.311,155.386
C03235=1064.326,141.394,421.704,172.540,29.314,155.386
C03236=1064.332,141.644,421.683,172.542,29.316,155.387
C03237=1064.338,141.893,421.662,172.544,29.319,155.387
C03238=1064.344,142.142,421.642,172.545,29.322,155.387
C03239=1064.350,142.426,421.618,172.548,29.325,155.388
C03240=1064.357,142.710,421.594,172.549,29.329,155.388
C03241=1064.364,142.994,421.570,172.551,29.332,155.389
C03242=1064.370,143.277,421.546,172.554,29.335,155.389
C03243=1064.376,143.526,421.525,172.555,29.338,155.390
C03244=1064.381,143.775,421.504,172.557,29.340,155.390
C03245=1064.388,144.025,421.482,172.559,29.343,155.391
C03246=1064.393,144.273,421.461,172.560,29.346,155.391
C03247=1064.399,144.523,421.440,172.562,29.349,155.391
C03248=1064.405,144.771,421.420,172.564,29.352,155.392
C03249=1064.411,145.020,421.399,172.565,29.354,155.392
C03250=1064.417,145.269,421.377,172.567,29.357,155.393
C03251=1064.422,145.518,421.356,172.569,29.360,155.393
C03252=1064.428,145.768,421.335,172.571,29.363,155.393
C03253=1064.434,146.016,421.314,172.573,29.365,155.394
C03254=1064.440,146.266,421.293,172.575,29.368,155.394
C03255=1064.445,146.515,421.272,172.576,29.371,155.395
C03256=1064.452,146.763,421.251,172.578,29.374,155.395
C03257=1064.457,147.013,421.230,172.580,29.376,155.396
C03258=1064.463,147.262,421.209,172.581,29.379,155.396
C03259=1064.470,147.511,421.187,172.583,29.382,155.396
C03260=1064.475,147.759,421.166,172.585,29.384,155.397
C03261=1064.481,148.009,421.145,172.586,29.387,155.397
C03262=1064.487,148.258,421.123,172.589,29.391,155.398
C03263=1064.493,148.507,421.102,172.591,29.393,155.398
C03264=1064.498,148.756,421.081,172.592,29.396,155.398
C03265=1064.504,149.005,421.060,172.594,29.399,155.399
C03266=1064.510,149.254,421.038,172.596,29.401,155.399
C03267=1064.516,149.503,421.017,172.597,29.404,155.400
C03268=1064.521,149.752,420.995,172.599,29.407,155.400
C03269=1064.527,150.001,420.975,172.601,29.410,155.401
C03270=1064.533,150.250,420.953,172.602,29.413,155.401
C03271=1064.539,150.499,420.932,172.605,29.416,155.401
C03272=1064.544,150.748,420.910,172.607,29.418,155.402
C03273=1064.550,150.997,420.888,172.608,29.421,155.402
C03274=1064.556,151.246,420.867,172.610,29.424,155.403
C03275=1064.561,151.495,420.846,172.612,29.427,155.403
C03276=1064.568,151.745,420.824,172.613,29.429,155.403
C03277=1064.573,151.993,420.803,172.615,29.433,155.404
C03278=1064.579,152.242,420.781,172.617,29.435,155.404
C03279=1064.585,152.491,420.760,172.619,29.438,155.405
C03280=1064.591,152.740,420.738,172.621,29.441,155.405
C03281=1064.596,152.989,420.717,172.623,29.444,155.406
C03282=1064.602,153.238,420.695,172.624,29.446,155.406
C03283=1064.608,153.487,420.673,172.626,29.449,155.406
C03284=1064.614,153.736,420.652,172.628,29.452,155.407
C03285=1064.620,153.986,420.631,172.629,29.455,155.407
C03286=1064.625,154.234,420.610,172.632,29.458,155.408
C03287=1064.631,154.483,420.588,172.634,29.461,155.408
C03288=1064.637,154.733,420.566,172.635,29.463,155.409
C03289=1064.642,154.981,420.545,172.637,29.466,155.409
C03290=1064.648,155.231,420.523,172.639,29.469,155.409
C03291=1064.654,155.479,420.502,172.640,29.471,155.410
C03292=1064.660,155.728,420.480,172.642,29.475,155.410
C03293=1064.666,155.978,420.458,172.645,29.478,155.411
C03294=1064.671,156.226,420.437,172.646,29.480,155.411
C03295=1064.678,156.475,420.414,172.648,29.483,155.412
C03296=1064.684,156.724,420.393,172.650,29.486,155.412
C03297=1064.689,156.973,420.371,172.651,29.488,155.412
C03298=1064.695,157.222,420.349,172.653,29.492,155.413
C03299=1064.701,157.471,420.328,172.656,29.494,155.413
C03300=1064.706,157.720,420.306,172.657,29.497,155.414
C03301=1064.712,157.969,420.284,172.659,29.500,155.414
C03302=1064.718,158.218,420.263,172.661,29.503,155.415
C03303=1064.724,158.502,420.238,172.663,29.506,155.415
C03304=1064.731,158.785,420.213,172.665,29.509,155.416
C03305=1064.738,159.068,420.188,172.667,29.512,155.416
C03306=1064.744,159.352,420.163,172.669,29.515,155.416
C03307=1064.750,159.601,420.141,172.671,29.518,155.417
C03308=1064.756,159.850,420.120,172.672,29.521,155.417
C03309=1064.761,160.099,420.098,172.675,29.524,155.418
C03310=1064.767,160.349,420.076,172.677,29.527,155.418
C03311=1064.774,160.597,420.054,172.678,29.530,155.419
C03312=1064.779,160.846,420.032,172.680,29.532,155.419
C03313=1064.785,161.095,420.010,172.682,29.535,155.419
C03314=1064.791,161.344,419.988,172.683,29.538,155.420
C03315=1064.796,161.593,419.966,172.686,29.541,155.420
C03316=1064.802,161.842,419.944,172.688,29.544,155.421
C03317=1064.808,162.091,419.922,172.689,29.547,155.421
C03318=1064.813,162.340,419.900,172.691,29.550,155.422
C03319=1064.818,162.589,419.877,172.693,29.553,155.422
C03320=1064.824,162.838,419.856,172.695,29.556,155.423
C03321=1064.829,163.087,419.834,172.697,29.559,155.423
C03322=1064.835,163.336,419.811,172.699,29.561,155.423
C03323=1064.841,163.584,419.790,172.700,29.565,155.424
C03324=1064.846,163.833,419.767,172.702,29.567,155.424
C03325=1064.852,164.083,419.744,172.705,29.570,155.425
C03326=1064.858,164.332,419.723,172.706,29.574,155.425
C03327=1064.863,164.580,419.700,172.708,29.576,155.426
C03328=1064.869,164.829,419.678,172.710,29.579,155.426
C03329=1064.875,165.078,419.656,172.711,29.582,155.427
C03330=1064.880,165.327,419.634,172.714,29.585,155.427
C03331=1064.886,165.576,419.612,172.716,29.588,155.427
C03332=1064.892,165.825,419.589,172.717,29.591,155.428
C03333=1064.897,166.074,419.567,172.719,29.594,155.428
C03334=1064.903,166.323,419.545,172.721,29.596,155.429
C03335=1064.908,166.572,419.523,172.723,29.600,155.429
C03336=1064.914,166.821,419.500,172.725,29.603,155.430
C03337=1064.919,167.070,419.478,172.727,29.605,155.430
C03338=1064.925,167.319,419.456,172.728,29.608,155.431
C03339=1064.931,167.568,419.433,172.730,29.611,155.431
C03340=1064.937,167.817,419.410,172.733,29.614,155.431
C03341=1064.943,168.066,419.389,172.734,29.617,155.432
C03342=1064.948,168.314,419.366,172.736,29.620,155.432
C03343=1064.953,168.564,419.344,172.738,29.623,155.433
C03344=1064.960,168.812,419.322,172.740,29.626,155.433
C03345=1064.965,169.062,419.299,172.742,29.629,155.434
C03346=1064.970,169.310,419.277,172.744,29.632,155.434
C03347=1064.976,169.559,419.254,172.745,29.634,155.435
C03348=1064.982,169.808,419.232,172.748,29.638,155.435
C03349=1064.988,170.057,419.209,172.750,29.640,155.435
C03350=1064.993,170.307,419.187,172.751,29.643,155.436
C03351=1065.000,170.555,419.165,172.753,29.646,155.436
C03352=1065.005,170.803,419.142,172.756,29.649,155.437
C03353=1065.010,171.053,419.120,172.757,29.652,155.437
C03354=1065.016,171.302,419.097,172.759,29.655,155.438
C03355=1065.023,171.550,419.075,172.761,29.658,155.438
C03356=1065.028,171.800,419.052,172.763,29.661,155.439
C03357=1065.034,172.049,419.029,172.765,29.663,155.439
C03358=1065.039,172.298,419.006,172.767,29.667,155.439
C03359=1065.045,172.546,418.984,172.768,29.669,155.440
C03360=1065.051,172.795,418.962,172.771,29.672,155.440
C03361=1065.057,173.044,418.939,172.773,29.676,155.441
C03362=1065.062,173.293,418.916,172.774,29.678,155.441
C03363=1065.068,173.542,418.895,172.777,29.681,155.442
C03364=1065.074,173.791,418.872,172.779,29.684,155.442
C03365=1065.080,174.040,418.849,172.780,29.687,155.443
C03366=1065.086,174.289,418.826,172.782,29.690,155.443
C03367=1065.092,174.572,418.800,172.785,29.693,155.443
C03368=1065.099,174.855,418.775,172.787,29.697,155.444
C03369=1065.106,175.138,418.749,172.789,29.700,155.445
C03370=1065.112,175.422,418.723,172.792,29.703,155.445
C03371=1065.118,175.670,418.700,172.793,29.706,155.445
C03372=1065.123,175.919,418.677,172.795,29.709,155.446
C03373=1065.129,176.168,418.655,172.798,29.712,155.446
C03374=1065.135,176.417,418.633,172.799,29.715,155.447
C03375=1065.141,176.666,418.610,172.801,29.717,155.447
C03376=1065.147,176.915,418.587,172.804,29.720,155.448
C03377=1065.152,177.163,418.564,172.805,29.724,155.448
C03378=1065.158,177.412,418.541,172.807,29.726,155.449
C03379=1065.165,177.661,418.519,172.810,29.729,155.449
C03380=1065.170,177.910,418.496,172.811,29.732,155.449
C03381=1065.176,178.159,418.473,172.813,29.735,155.450
C03382=1065.182,178.408,418.450,172.815,29.738,155.450
C03383=1065.187,178.657,418.428,172.817,29.741,155.451
C03384=1065.194,178.906,418.405,172.819,29.744,155.451
C03385=1065.199,179.155,418.382,172.821,29.747,155.452
C03386=1065.205,179.404,418.359,172.824,29.749,155.452
C03387=1065.211,179.653,418.336,172.825,29.752,155.452
C03388=1065.217,179.902,418.313,172.827,29.755,155.453
C03389=1065.223,180.151,418.290,172.830,29.758,155.453
C03390=1065.229,180.400,418.268,172.831,29.761,155.454
C03391=1065.235,180.648,418.245,172.833,29.764,155.454
C03392=1065.241,180.897,418.222,172.836,29.767,155.455
C03393=1065.247,181.146,418.198,172.837,29.770,155.455
C03394=1065.253,181.394,418.175,172.840,29.773,155.455
C03395=1065.258,181.643,418.152,172.842,29.776,155.456
C03396=1065.264,181.892,418.130,172.843,29.778,155.456
C03397=1065.271,182.141,418.107,172.846,29.781,155.457
C03398=1065.276,182.390,418.084,172.848,29.784,155.457
C03399=1065.283,182.639,418.061,172.849,29.787,155.458
C03400=1065.288,182.888,418.038,172.852,29.790,155.458
C03401=1065.294,183.137,418.015,172.854,29.793,155.459
C03402=1065.300,183.386,417.992,172.855,29.796,155.459
C03403=1065.306,183.634,417.968,172.858,29.799,155.460
C03404=1065.312,183.883,417.945,172.860,29.802,155.460
C03405=1065.318,184.132,417.923,172.862,29.804,155.460
C03406=1065.324,184.381,417.900,172.864,29.808,155.461
C03407=1065.330,184.630,417.877,172.866,29.810,155.461
C03408=1065.335,184.879,417.853,172.868,29.814,155.462
C03409=1065.341,185.128,417.830,172.870,29.816,155.462
C03410=1065.347,185.377,417.807,172.872,29.820,155.463
C03411=1065.352,185.626,417.783,172.875,29.823,155.463
C03412=1065.358,185.874,417.759,172.876,29.826,155.464
C03413=1065.364,186.123,417.737,172.878,29.828,155.464
C03414=1065.369,186.372,417.713,172.881,29.832,155.465
C03415=1065.375,186.621,417.689,172.882,29.835,155.465
C03416=1065.380,186.869,417.666,172.885,29.838,155.465
C03417=1065.385,187.119,417.643,172.887,29.841,155.466
C03418=1065.391,187.367,417.619,172.888,29.844,155.466
C03419=1065.397,187.616,417.596,172.891,29.847,155.467
C03420=1065.402,187.865,417.573,172.893,29.850,155.467
C03421=1065.409,188.114,417.549,172.894,29.853,155.468
C03422=1065.414,188.363,417.526,172.897,29.856,155.468
C03423=1065.420,188.612,417.501,172.899,29.859,155.469
C03424=1065.426,188.860,417.479,172.901,29.863,155.469
C03425=1065.431,189.109,417.456,172.903,29.865,155.470
C03426=1065.437,189.358,417.431,172.905,29.869,155.470
C03427=1065.442,189.607,417.408,172.907,29.872,155.471
C03428=1065.448,189.855,417.384,172.909,29.875,155.471
C03429=1065.454,190.105,417.361,172.912,29.878,155.472
C03430=1065.460,190.353,417.337,172.913,29.881,155.472
C03431=1065.466,190.636,417.310,172.916,29.884,155.473
C03432=1065.473,190.919,417.284,172.918,29.887,155.473
C03433=1065.479,191.202,417.256,172.920,29.891,155.474
C03434=1065.486,191.484,417.230,172.923,29.895,155.474
C03435=1065.491,191.734,417.206,172.925,29.898,155.475
C03436=1065.497,191.982,417.183,172.927,29.901,155.475
C03437=1065.503,192.231,417.160,172.929,29.904,155.476
C03438=1065.508,192.479,417.135,172.932,29.907,155.476
C03439=1065.514,192.728,417.111,172.933,29.910,155.477
C03440=1065.519,192.978,417.088,172.935,29.913,155.477
C03441=1065.525,193.226,417.064,172.938,29.916,155.478
C03442=1065.531,193.475,417.041,172.939,29.919,155.478
C03443=1065.537,193.724,417.017,172.942,29.922,155.479
C03444=1065.543,193.972,416.993,172.944,29.925,155.479
C03445=1065.548,194.222,416.969,172.946,29.929,155.480
C03446=1065.554,194.470,416.946,172.948,29.932,155.480
C03447=1065.560,194.719,416.921,172.951,29.935,155.480
C03448=1065.566,194.968,416.898,172.952,29.938,155.481
C03449=1065.572,195.216,416.874,172.954,29.941,155.481
C03450=1065.577,195.465,416.850,172.957,29.944,155.482
C03451=1065.583,195.714,416.827,172.958,29.947,155.482
C03452=1065.589,195.963,416.803,172.961,29.950,155.483
C03453=1065.595,196.211,416.779,172.963,29.953,155.483
C03454=1065.601,196.461,416.754,172.965,29.956,155.484
C03455=1065.606,196.710,416.731,172.967,29.959,155.484
C03456=1065.612,196.958,416.707,172.970,29.962,155.485
C03457=1065.618,197.207,416.683,172.971,29.965,155.485
C03458=1065.624,197.456,416.659,172.974,29.968,155.486
C03459=1065.630,197.704,416.635,172.976,29.971,155.486
C03460=1065.635,197.954,416.611,172.978,29.975,155.487
C03461=1065.641,198.202,416.588,172.980,29.978,155.487
C03462=1065.647,198.450,416.564,172.983,29.981,155.488
C03463=1065.653,198.700,416.539,172.985,29.984,155.488
C03464=1065.659,198.948,416.516,172.987,29.987,155.489
C03465=1065.665,199.197,416.491,172.989,29.990,155.489
C03466=1065.671,199.446,416.468,172.992,29.993,155.489
C03467=1065.676,199.695,416.444,172.993,29.996,155.490
C03468=1065.683,199.944,416.420,172.996,29.999,155.490
C03469=1065.688,200.192,416.396,172.998,30.002,155.491
C03470=1065.694,200.441,416.372,173.000,30.006,155.491
C03471=1065.700,200.690,416.347,173.002,30.008,155.492
C03472=1065.706,200.938,416.324,173.005,30.012,155.492
C03473=1065.712,201.187,416.299,173.006,30.014,155.493
C03474=1065.717,201.436,416.275,173.009,30.018,155.493
C03475=1065.723,201.684,416.251,173.011,30.021,155.494
C03476=1065.729,201.934,416.226,173.013,30.024,155.494
C03477=1065.735,202.182,416.203,173.015,30.027,155.495
C03478=1065.741,202.431,416.178,173.018,30.031,155.495
C03479=1065.747,202.680,416.154,173.019,30.033,155.496
C03480=1065.753,202.928,416.130,173.022,30.037,155.496
C03481=1065.758,203.177,416.106,173.024,30.040,155.497
C03482=1065.764,203.426,416.081,173.026,30.043,155.497
C03483=1065.770,203.675,416.057,173.028,30.046,155.498
C03484=1065.775,203.924,416.032,173.031,30.049,155.498
C03485=1065.781,204.172,416.009,173.033,30.053,155.499
C03486=1065.787,204.421,415.983,173.035,30.056,155.499
C03487=1065.793,204.669,415.959,173.037,30.059,155.500
C03488=1065.798,204.919,415.935,173.040,30.062,155.500
C03489=1065.804,205.167,415.910,173.042,30.065,155.501
C03490=1065.810,205.416,415.886,173.044,30.069,155.501
C03491=1065.816,205.665,415.862,173.047,30.072,155.502
C03492=1065.822,205.913,415.837,173.048,30.075,155.502
C03493=1065.827,206.162,415.812,173.051,30.078,155.503
C03494=1065.833,206.411,415.788,173.053,30.081,155.503
C03495=1065.857,207.456,415.685,173.209,30.159,155.508
C03496=1065.863,207.676,415.663,173.211,30.163,155.509
C03497=1065.868,207.897,415.641,173.213,30.166,155.510
C03498=1065.874,208.116,415.618,173.214,30.170,155.510
C03499=1065.879,208.336,415.596,173.216,30.173,155.511
C03500=1065.884,208.556,415.574,173.218,30.177,155.512
C03501=1065.889,208.776,415.551,173.219,30.181,155.512
C03502=1065.894,208.995,415.528,173.221,30.184,155.513
C03503=1065.900,209.215,415.506,173.223,30.188,155.513
C03504=1065.905,209.464,415.481,173.225,30.192,155.514
C03505=1065.911,209.712,415.456,173.227,30.196,155.515
C03506=1065.917,209.961,415.431,173.229,30.200,155.516
C03507=1065.923,210.210,415.405,173.231,30.204,155.516
C03508=1065.930,210.458,415.380,173.233,30.208,155.517
C03509=1065.936,210.707,415.355,173.234,30.212,155.518
C03510=1065.941,210.956,415.329,173.237,30.216,155.518
C03511=1065.948,211.205,415.303,173.239,30.221,155.519
C03512=1065.953,211.453,415.278,173.240,30.224,155.520
C03513=1065.960,211.701,415.252,173.243,30.229,155.521
C03514=1065.965,211.950,415.226,173.245,30.233,155.521
C03515=1065.971,212.198,415.201,173.247,30.237,155.522
C03516=1065.978,212.447,415.176,173.249,30.241,155.523
C03517=1065.983,212.696,415.150,173.250,30.245,155.523
C03518=1065.989,212.945,415.124,173.253,30.249,155.524
C03519=1065.995,213.193,415.099,173.255,30.253,155.525
C03520=1066.001,213.442,415.073,173.256,30.257,155.526
C03521=1066.007,213.691,415.048,173.259,30.261,155.526
C03522=1066.013,213.938,415.022,173.261,30.265,155.527
C03523=1066.019,214.187,414.996,173.263,30.269,155.528
C03524=1066.025,214.436,414.971,173.265,30.274,155.528
C03525=1066.030,214.685,414.945,173.266,30.277,155.529
C03526=1066.036,214.934,414.920,173.269,30.282,155.530
C03527=1066.043,215.182,414.894,173.271,30.286,155.531
C03528=1066.048,215.431,414.868,173.272,30.290,155.531
C03529=1066.055,215.679,414.842,173.275,30.294,155.532
C03530=1066.060,215.928,414.816,173.277,30.298,155.533
C03531=1066.067,216.176,414.790,173.279,30.302,155.533
C03532=1066.072,216.425,414.764,173.281,30.306,155.534
C03533=1066.078,216.674,414.739,173.282,30.310,155.535
C03534=1066.085,216.922,414.713,173.285,30.314,155.535
C03535=1066.090,217.171,414.687,173.287,30.318,155.536
C03536=1066.096,217.420,414.662,173.289,30.322,155.537
C03537=1066.102,217.668,414.635,173.291,30.327,155.538
C03538=1066.108,217.917,414.610,173.294,30.330,155.538
C03539=1066.114,218.166,414.584,173.295,30.334,155.539
C03540=1066.120,218.414,414.558,173.297,30.339,155.540
C03541=1066.126,218.663,414.532,173.300,30.342,155.540
C03542=1066.132,218.911,414.507,173.301,30.347,155.541
C03543=1066.138,219.160,414.480,173.304,30.351,155.542
C03544=1066.144,219.409,414.455,173.306,30.354,155.542
C03545=1066.150,219.657,414.428,173.307,30.359,155.543
C03546=1066.156,219.906,414.403,173.310,30.363,155.544
C03547=1066.162,220.154,414.376,173.312,30.366,155.545
C03548=1066.168,220.403,414.351,173.314,30.371,155.545
C03549=1066.174,220.651,414.324,173.316,30.375,155.546
C03550=1066.180,220.900,414.299,173.318,30.378,155.547
C03551=1066.187,221.148,414.272,173.320,30.383,155.547
C03552=1066.191,221.371,414.249,173.322,30.386,155.548
C03553=1066.196,221.593,414.226,173.323,30.390,155.549
C03554=1066.202,221.815,414.202,173.326,30.394,155.549
C03555=1066.207,222.037,414.179,173.328,30.397,155.550
C03556=1066.213,222.259,414.156,173.330,30.401,155.551
C03557=1066.218,222.482,414.132,173.331,30.404,155.551
C03558=1066.223,222.703,414.109,173.333,30.408,155.552
C03559=1066.228,222.926,414.085,173.336,30.412,155.552
C03560=1066.235,223.174,414.059,173.337,30.416,155.553
C03561=1066.240,223.422,414.033,173.339,30.420,155.554
C03562=1066.246,223.672,414.006,173.342,30.424,155.555
C03563=1066.253,223.920,413.980,173.343,30.428,155.555
C03564=1066.259,224.168,413.954,173.346,30.432,155.556
C03565=1066.264,224.417,413.928,173.347,30.436,155.557
C03566=1066.270,224.665,413.901,173.350,30.440,155.557
C03567=1066.276,224.914,413.875,173.352,30.444,155.558
C03568=1066.282,225.162,413.849,173.354,30.448,155.559
C03569=1066.288,225.411,413.822,173.356,30.452,155.560
C03570=1066.294,225.660,413.795,173.359,30.456,155.560
C03571=1066.301,225.908,413.769,173.360,30.460,155.561
C03572=1066.306,226.157,413.743,173.363,30.464,155.562
C03573=1066.312,226.405,413.717,173.365,30.468,155.562
C03574=1066.318,226.654,413.690,173.367,30.472,155.563
C03575=1066.324,226.902,413.664,173.369,30.476,155.564
C03576=1066.330,227.151,413.638,173.372,30.480,155.564
C03577=1066.336,227.400,413.611,173.373,30.484,155.565
C03578=1066.342,227.648,413.584,173.376,30.488,155.566
C03579=1066.347,227.896,413.558,173.378,30.492,155.566
C03580=1066.354,228.145,413.532,173.379,30.496,155.567
C03581=1066.360,228.394,413.505,173.382,30.500,155.568
C03582=1066.366,228.642,413.478,173.384,30.504,155.569
C03583=1066.372,228.891,413.452,173.386,30.508,155.569
C03584=1066.378,229.139,413.426,173.389,30.512,155.570
C03585=1066.384,229.388,413.399,173.391,30.516,155.571
C03586=1066.390,229.636,413.372,173.393,30.520,155.571
C03587=1066.396,229.885,413.346,173.395,30.524,155.572
C03588=1066.402,230.133,413.319,173.398,30.528,155.573
C03589=1066.408,230.382,413.292,173.399,30.532,155.573
C03590=1066.414,230.631,413.266,173.402,30.536,155.574
C03591=1066.420,230.879,413.239,173.404,30.540,155.575
C03592=1066.426,231.127,413.212,173.406,30.544,155.575
C03593=1066.432,231.376,413.185,173.408,30.548,155.576
C03594=1066.438,231.625,413.159,173.411,30.552,155.577
C03595=1066.443,231.873,413.132,173.412,30.556,155.578
C03596=1066.449,232.121,413.105,173.415,30.560,155.578
C03597=1066.456,232.370,413.078,173.417,30.564,155.579
C03598=1066.461,232.619,413.052,173.419,30.568,155.580
C03599=1066.467,232.867,413.025,173.421,30.572,155.580
C03600=1066.474,233.116,412.997,173.424,30.576,155.581
C03601=1066.480,233.364,412.971,173.425,30.580,155.582
C03602=1066.485,233.612,412.944,173.428,30.584,155.583
C03603=1066.491,233.861,412.917,173.430,30.588,155.583
C03604=1066.497,234.110,412.890,173.432,30.592,155.584
C03605=1066.503,234.358,412.864,173.434,30.596,155.585
C03606=1066.509,234.606,412.836,173.437,30.600,155.585
C03607=1066.515,234.855,412.809,173.439,30.604,155.586
C03608=1066.520,235.074,412.786,173.441,30.608,155.587
C03609=1066.525,235.292,412.762,173.443,30.611,155.587
C03610=1066.531,235.509,412.738,173.445,30.614,155.588
C03611=1066.536,235.727,412.714,173.446,30.618,155.589
C03612=1066.541,235.946,412.691,173.449,30.621,155.589
C03613=1066.547,236.164,412.667,173.451,30.625,155.590
C03614=1066.552,236.381,412.643,173.453,30.629,155.590
C03615=1066.556,236.600,412.619,173.454,30.632,155.591
C03616=1066.562,236.848,412.592,173.457,30.636,155.592
C03617=1066.569,237.097,412.565,173.460,30.640,155.592
C03618=1066.575,237.345,412.538,173.461,30.644,155.593
C03619=1066.581,237.594,412.511,173.464,30.648,155.594
C03620=1066.587,237.842,412.484,173.466,30.652,155.594
C03621=1066.592,238.090,412.456,173.468,30.656,155.595
C03622=1066.599,238.339,412.429,173.470,30.660,155.596
C03623=1066.604,238.588,412.403,173.473,30.664,155.597
C03624=1066.611,238.836,412.375,173.475,30.668,155.597
C03625=1066.617,239.084,412.348,173.477,30.672,155.598
C03626=1066.622,239.332,412.320,173.480,30.676,155.599
C03627=1066.629,239.582,412.293,173.482,30.680,155.599
C03628=1066.635,239.829,412.266,173.484,30.684,155.600
C03629=1066.641,240.078,412.239,173.487,30.688,155.601
C03630=1066.646,240.326,412.211,173.489,30.692,155.601
C03631=1066.653,240.575,412.184,173.491,30.696,155.602
C03632=1066.659,240.823,412.156,173.493,30.700,155.603
C03633=1066.665,241.072,412.129,173.496,30.703,155.603
C03634=1066.670,241.320,412.101,173.498,30.708,155.604
C03635=1066.676,241.569,412.075,173.500,30.712,155.605
C03636=1066.683,241.817,412.047,173.503,30.715,155.605
C03637=1066.689,242.066,412.020,173.504,30.720,155.606
C03638=1066.695,242.314,411.992,173.507,30.724,155.607
C03639=1066.701,242.563,411.965,173.510,30.727,155.608
C03640=1066.706,242.811,411.937,173.512,30.731,155.608
